LIN {X 0,Y 468.343,Z 264.353,A -85,B 0,C 180,E1 -7622.765,E2 -7622.765} C_VEL
LIN {X 0,Y 467.925,Z 273.797,A -85,B 0,C 180,E1 -7626.076,E2 -7626.076} C_VEL
LIN {X 0,Y 467.627,Z 283.274,A -85,B 0,C 180,E1 -7629.318,E2 -7629.318} C_VEL
LIN {X 0,Y 467.347,Z 292.793,A -85,B 0,C 180,E1 -7632.497,E2 -7632.497} C_VEL
LIN {X 0,Y 467.211,Z 299.063,A -85,B 0,C 180,E1 -7634.57,E2 -7634.57} C_VEL
LIN {X 0,Y 469.771,Z 314.339,A -85,B 0,C 180,E1 -7635.072,E2 -7635.072} C_VEL
LIN {X 0,Y 470.153,Z 319.57,A -85,B 0,C 180,E1 -7635.278,E2 -7635.278} C_VEL
LIN {X 0,Y 469.716,Z 331.244,A -85,B 0,C 180,E1 -7635.818,E2 -7635.818} C_VEL
LIN {X 0,Y 469.238,Z 342.474,A -85,B 0,C 180,E1 -7636.499,E2 -7636.499} C_VEL
LIN {X 0,Y 468.797,Z 353.368,A -85,B 0,C 180,E1 -7637.336,E2 -7637.336} C_VEL
LIN {X 0,Y 468.377,Z 363.596,A -85,B 0,C 180,E1 -7638.313,E2 -7638.313} C_VEL
LIN {X 0,Y 467.886,Z 372.785,A -85,B 0,C 180,E1 -7639.397,E2 -7639.397} C_VEL
LIN {X 0,Y 467.447,Z 381.688,A -85,B 0,C 180,E1 -7640.699,E2 -7640.699} C_VEL
LIN {X 0,Y 467.092,Z 388.849,A -85,B 0,C 180,E1 -7642,E2 -7642} C_VEL
LIN {X 0,Y 466.87,Z 395.224,A -85,B 0,C 180,E1 -7643.479,E2 -7643.479} C_VEL
LIN {X 0,Y 466.784,Z 399.677,A -85,B 0,C 180,E1 -7644.817,E2 -7644.817} C_VEL
LIN {X 0,Y 466.663,Z 401.958,A -85,B 0,C 180,E1 -7645.682,E2 -7645.682} C_VEL
LIN {X 0,Y 466.695,Z 403.807,A -85,B 0,C 180,E1 -7646.547,E2 -7646.547} C_VEL
LIN {X 0,Y 466.646,Z 405.193,A -85,B 0,C 180,E1 -7647.41,E2 -7647.41} C_VEL
LIN {X 0,Y 466.589,Z 406.785,A -85,B 0,C 180,E1 -7649.137,E2 -7649.137} C_VEL
LIN {X 0,Y 466.57,Z 407,A -85,B 0,C 180,E1 -7650,E2 -7650} C_VEL
LIN {X 0,Y 466.589,Z 406.786,A -85,B 0,C 180,E1 -7650.863,E2 -7650.863} C_VEL
LIN {X 0,Y 466.646,Z 405.195,A -85,B 0,C 180,E1 -7652.59,E2 -7652.59} C_VEL
LIN {X 0,Y 466.695,Z 403.81,A -85,B 0,C 180,E1 -7653.454,E2 -7653.454} C_VEL
LIN {X 0,Y 466.703,Z 400.895,A -85,B 0,C 180,E1 -7654.751,E2 -7654.751} C_VEL
LIN {X 0,Y 466.841,Z 396.947,A -85,B 0,C 180,E1 -7656.049,E2 -7656.049} C_VEL
LIN {X 0,Y 466.998,Z 390.874,A -85,B 0,C 180,E1 -7657.567,E2 -7657.567} C_VEL
LIN {X 0,Y 467.35,Z 384.234,A -85,B 0,C 180,E1 -7658.867,E2 -7658.867} C_VEL
LIN {X 0,Y 467.741,Z 375.991,A -85,B 0,C 180,E1 -7660.169,E2 -7660.169} C_VEL
LIN {X 0,Y 468.137,Z 367.516,A -85,B 0,C 180,E1 -7661.255,E2 -7661.255} C_VEL
LIN {X 0,Y 468.646,Z 357.189,A -85,B 0,C 180,E1 -7662.32,E2 -7662.32} C_VEL
LIN {X 0,Y 469.084,Z 345.563,A -85,B 0,C 180,E1 -7663.285,E2 -7663.285} C_VEL
LIN {X 0,Y 469.647,Z 333.231,A -85,B 0,C 180,E1 -7664.074,E2 -7664.074} C_VEL
LIN {X 0,Y 470.102,Z 320.858,A -85,B 0,C 180,E1 -7664.668,E2 -7664.668} C_VEL
LIN {X 0,Y 469.911,Z 315.479,A -85,B 0,C 180,E1 -7664.882,E2 -7664.882} C_VEL
LIN {X 0,Y 467.86,Z 303.142,A -85,B 0,C 180,E1 -7665.307,E2 -7665.307} C_VEL
LIN {X 0,Y 467.212,Z 298.992,A -85,B 0,C 180,E1 -7665.43,E2 -7665.43} C_VEL
LIN {X 0,Y 467.478,Z 289.113,A -85,B 0,C 180,E1 -7668.713,E2 -7668.713} C_VEL
LIN {X 0,Y 467.753,Z 279.15,A -85,B 0,C 180,E1 -7672.063,E2 -7672.063} C_VEL
LIN {X 0,Y 468.076,Z 269.794,A -85,B 0,C 180,E1 -7675.298,E2 -7675.298} C_VEL
LIN {X 0,Y 468.411,Z 261.608,A -85,B 0,C 180,E1 -7678.205,E2 -7678.205} C_VEL
LIN {X 0,Y 468.861,Z 252.156,A -85,B 0,C 180,E1 -7681.644,E2 -7681.644} C_VEL
LIN {X 0,Y 469.23,Z 244.096,A -85,B 0,C 180,E1 -7684.692,E2 -7684.692} C_VEL
LIN {X 0,Y 469.305,Z 240.672,A -85,B 0,C 180,E1 -7686.034,E2 -7686.034} C_VEL
LIN {X 0,Y 468.317,Z 234.357,A -85,B 0,C 180,E1 -7688.706,E2 -7688.706} C_VEL
LIN {X 0,Y 467.579,Z 230.247,A -85,B 0,C 180,E1 -7690.619,E2 -7690.619} C_VEL
LIN {X 0,Y 467.557,Z 230.25,A -85,B 0,C 180,E1 -7693.745,E2 -7693.745} C_VEL
LIN {X 0,Y 467.55,Z 230.244,A -85,B 0,C 180,E1 -7696.255,E2 -7696.255} C_VEL
LIN {X 0,Y 467.562,Z 230.24,A -85,B 0,C 180,E1 -7699.734,E2 -7699.734} C_VEL
LIN {X 0,Y 467.546,Z 230.246,A -85,B 0,C 180,E1 -7702.815,E2 -7702.815} C_VEL
LIN {X 0,Y 467.59,Z 230.241,A -85,B 0,C 180,E1 -7706.212,E2 -7706.212} C_VEL
LIN {X 0,Y 467.57,Z 230.242,A -85,B 0,C 180,E1 -7709.266,E2 -7709.266} C_VEL
LIN {X 0,Y 467.553,Z 230.247,A -85,B 0,C 180,E1 -7712.482,E2 -7712.482} C_VEL
LIN {X 0,Y 467.563,Z 230.241,A -85,B 0,C 180,E1 -7715.11,E2 -7715.11} C_VEL
LIN {X 0,Y 467.539,Z 230.249,A -85,B 0,C 180,E1 -7717.926,E2 -7717.926} C_VEL
LIN {X 0,Y 467.627,Z 230.236,A -85,B 0,C 180,E1 -7720.692,E2 -7720.692} C_VEL
LIN {X 0,Y 467.654,Z 230.234,A -85,B 0,C 180,E1 -7724.115,E2 -7724.115} C_VEL
LIN {X 0,Y 467.652,Z 230.233,A -85,B 0,C 180,E1 -7727.646,E2 -7727.646} C_VEL
LIN {X 0,Y 467.665,Z 230.232,A -85,B 0,C 180,E1 -7731.357,E2 -7731.357} C_VEL
LIN {X 0,Y 467.739,Z 230.222,A -85,B 0,C 180,E1 -7733.963,E2 -7733.963} C_VEL
LIN {X 0,Y 467.864,Z 230.206,A -85,B 0,C 180,E1 -7737.417,E2 -7737.417} C_VEL
LIN {X 0,Y 467.853,Z 230.207,A -85,B 0,C 180,E1 -7740,E2 -7740} C_VEL
LIN {X 0,Y 467.825,Z 230.208,A -85,B 0,C 180,E1 -7742.583,E2 -7742.583} C_VEL
LIN {X 0,Y 467.737,Z 230.221,A -85,B 0,C 180,E1 -7746.038,E2 -7746.038} C_VEL
LIN {X 0,Y 467.674,Z 230.231,A -85,B 0,C 180,E1 -7748.643,E2 -7748.643} C_VEL
LIN {X 0,Y 467.661,Z 230.231,A -85,B 0,C 180,E1 -7752.145,E2 -7752.145} C_VEL
LIN {X 0,Y 467.642,Z 230.232,A -85,B 0,C 180,E1 -7755.695,E2 -7755.695} C_VEL
LIN {X 0,Y 467.625,Z 230.235,A -85,B 0,C 180,E1 -7759.308,E2 -7759.308} C_VEL
LIN {X 0,Y 467.539,Z 230.246,A -85,B 0,C 180,E1 -7762.074,E2 -7762.074} C_VEL
LIN {X 0,Y 467.59,Z 230.241,A -85,B 0,C 180,E1 -7764.888,E2 -7764.888} C_VEL
LIN {X 0,Y 467.565,Z 230.243,A -85,B 0,C 180,E1 -7767.773,E2 -7767.773} C_VEL
LIN {X 0,Y 467.549,Z 230.244,A -85,B 0,C 180,E1 -7771.04,E2 -7771.04} C_VEL
LIN {X 0,Y 467.574,Z 230.241,A -85,B 0,C 180,E1 -7773.789,E2 -7773.789} C_VEL
LIN {X 0,Y 467.534,Z 230.248,A -85,B 0,C 180,E1 -7776.962,E2 -7776.962} C_VEL
LIN {X 0,Y 467.574,Z 230.242,A -85,B 0,C 180,E1 -7779.953,E2 -7779.953} C_VEL
LIN {X 0,Y 467.564,Z 230.245,A -85,B 0,C 180,E1 -7782.563,E2 -7782.563} C_VEL
LIN {X 0,Y 467.569,Z 230.24,A -85,B 0,C 180,E1 -7785.052,E2 -7785.052} C_VEL
LIN {X 0,Y 467.576,Z 230.241,A -85,B 0,C 180,E1 -7788.596,E2 -7788.596} C_VEL
LIN {X 0,Y 467.565,Z 230.243,A -85,B 0,C 180,E1 -7791.955,E2 -7791.955} C_VEL
LIN {X 0,Y 467.429,Z 230.261,A -85,B 0,C 180,E1 -7795.155,E2 -7795.155} C_VEL
LIN {X 0,Y 467.198,Z 230.291,A -85,B 0,C 180,E1 -7797.395,E2 -7797.395} C_VEL
LIN {X 0,Y 467.077,Z 232.866,A -85,B 0,C 180,E1 -7800.228,E2 -7800.228} C_VEL
LIN {X 0,Y 467.014,Z 235.784,A -85,B 0,C 180,E1 -7803.162,E2 -7803.162} C_VEL
LIN {X 0,Y 466.95,Z 238.685,A -85,B 0,C 180,E1 -7806.022,E2 -7806.022} C_VEL
LIN {X 0,Y 466.898,Z 241.727,A -85,B 0,C 180,E1 -7808.949,E2 -7808.949} C_VEL
LIN {X 0,Y 466.894,Z 244.613,A -85,B 0,C 180,E1 -7811.572,E2 -7811.572} C_VEL
LIN {X 0,Y 466.87,Z 247.359,A -85,B 0,C 180,E1 -7813.911,E2 -7813.911} C_VEL
LIN {X 0,Y 466.79,Z 248.655,A -85,B 0,C 180,E1 -7814.261,E2 -7814.261} C_VEL
LIN {X 0,Y 466.58,Z 251.014,A -85,B 0,C 180,E1 -7814.532,E2 -7814.532} C_VEL
LIN {X 0,Y 466.15,Z 255.079,A -85,B 0,C 180,E1 -7814.785,E2 -7814.785} C_VEL
LIN {X 0,Y 463.561,Z 272.449,A -85,B 0,C 180,E1 -7815.439,E2 -7815.439} C_VEL
LIN {X 0,Y 463.282,Z 275.826,A -85,B 0,C 180,E1 -7815.608,E2 -7815.608} C_VEL
LIN {X 0,Y 462.831,Z 287.027,A -85,B 0,C 180,E1 -7816.291,E2 -7816.291} C_VEL
LIN {X 0,Y 462.369,Z 298.125,A -85,B 0,C 180,E1 -7817.156,E2 -7817.156} C_VEL
LIN {X 0,Y 461.823,Z 308.332,A -85,B 0,C 180,E1 -7818.144,E2 -7818.144} C_VEL
LIN {X 0,Y 461.343,Z 317.483,A -85,B 0,C 180,E1 -7819.245,E2 -7819.245} C_VEL
LIN {X 0,Y 460.871,Z 326.359,A -85,B 0,C 180,E1 -7820.565,E2 -7820.565} C_VEL
LIN {X 0,Y 460.435,Z 333.504,A -85,B 0,C 180,E1 -7821.883,E2 -7821.883} C_VEL
LIN {X 0,Y 460.182,Z 339.823,A -85,B 0,C 180,E1 -7823.373,E2 -7823.373} C_VEL
LIN {X 0,Y 459.847,Z 344.308,A -85,B 0,C 180,E1 -7824.738,E2 -7824.738} C_VEL
LIN {X 0,Y 459.919,Z 346.57,A -85,B 0,C 180,E1 -7825.618,E2 -7825.618} C_VEL
LIN {X 0,Y 459.824,Z 348.421,A -85,B 0,C 180,E1 -7826.495,E2 -7826.495} C_VEL
LIN {X 0,Y 459.781,Z 349.815,A -85,B 0,C 180,E1 -7827.372,E2 -7827.372} C_VEL
LIN {X 0,Y 459.567,Z 351.426,A -85,B 0,C 180,E1 -7829.124,E2 -7829.124} C_VEL
LIN {X 0,Y 459.55,Z 351.66,A -85,B 0,C 180,E1 -7830,E2 -7830} C_VEL
LIN {X 0,Y 459.642,Z 350.892,A -85,B 0,C 180,E1 -7831.752,E2 -7831.752} C_VEL
LIN {X 0,Y 459.781,Z 349.928,A -85,B 0,C 180,E1 -7832.628,E2 -7832.628} C_VEL
LIN {X 0,Y 459.823,Z 348.583,A -85,B 0,C 180,E1 -7833.505,E2 -7833.505} C_VEL
LIN {X 0,Y 459.903,Z 345.741,A -85,B 0,C 180,E1 -7834.821,E2 -7834.821} C_VEL
LIN {X 0,Y 460.044,Z 341.884,A -85,B 0,C 180,E1 -7836.139,E2 -7836.139} C_VEL
LIN {X 0,Y 460.253,Z 336.906,A -85,B 0,C 180,E1 -7837.458,E2 -7837.458} C_VEL
LIN {X 0,Y 460.598,Z 330.632,A -85,B 0,C 180,E1 -7838.777,E2 -7838.777} C_VEL
LIN {X 0,Y 461.004,Z 322.776,A -85,B 0,C 180,E1 -7840.097,E2 -7840.097} C_VEL
LIN {X 0,Y 461.527,Z 314.755,A -85,B 0,C 180,E1 -7841.195,E2 -7841.195} C_VEL
LIN {X 0,Y 462,Z 304.971,A -85,B 0,C 180,E1 -7842.296,E2 -7842.296} C_VEL
LIN {X 0,Y 462.475,Z 295.336,A -85,B 0,C 180,E1 -7843.176,E2 -7843.176} C_VEL
LIN {X 0,Y 462.937,Z 284.671,A -85,B 0,C 180,E1 -7843.961,E2 -7843.961} C_VEL
LIN {X 0,Y 463.391,Z 272.342,A -85,B 0,C 180,E1 -7844.66,E2 -7844.66} C_VEL
LIN {X 0,Y 463.563,Z 264.842,A -85,B 0,C 180,E1 -7844.998,E2 -7844.998} C_VEL
LIN {X 0,Y 460.782,Z 252.445,A -85,B 0,C 180,E1 -7845.514,E2 -7845.514} C_VEL
LIN {X 0,Y 459.861,Z 248.614,A -85,B 0,C 180,E1 -7845.671,E2 -7845.671} C_VEL
LIN {X 0,Y 459.83,Z 245.097,A -85,B 0,C 180,E1 -7848.721,E2 -7848.721} C_VEL
LIN {X 0,Y 459.836,Z 242.04,A -85,B 0,C 180,E1 -7851.519,E2 -7851.519} C_VEL
LIN {X 0,Y 459.903,Z 239.086,A -85,B 0,C 180,E1 -7854.368,E2 -7854.368} C_VEL
LIN {X 0,Y 459.989,Z 235.815,A -85,B 0,C 180,E1 -7857.605,E2 -7857.605} C_VEL
LIN {X 0,Y 460.045,Z 233.208,A -85,B 0,C 180,E1 -7860.274,E2 -7860.274} C_VEL
LIN {X 0,Y 460.081,Z 231.215,A -85,B 0,C 180,E1 -7862.32,E2 -7862.32} C_VEL
LIN {X 0,Y 460.428,Z 231.131,A -85,B 0,C 180,E1 -7865.453,E2 -7865.453} C_VEL
LIN {X 0,Y 460.52,Z 231.122,A -85,B 0,C 180,E1 -7868.734,E2 -7868.734} C_VEL
LIN {X 0,Y 460.52,Z 231.12,A -85,B 0,C 180,E1 -7871.6,E2 -7871.6} C_VEL
LIN {X 0,Y 460.514,Z 231.12,A -85,B 0,C 180,E1 -7874.589,E2 -7874.589} C_VEL
LIN {X 0,Y 460.506,Z 231.124,A -85,B 0,C 180,E1 -7877.816,E2 -7877.816} C_VEL
LIN {X 0,Y 460.534,Z 231.119,A -85,B 0,C 180,E1 -7881.104,E2 -7881.104} C_VEL
LIN {X 0,Y 460.511,Z 231.121,A -85,B 0,C 180,E1 -7884.554,E2 -7884.554} C_VEL
LIN {X 0,Y 460.532,Z 231.122,A -85,B 0,C 180,E1 -7887.715,E2 -7887.715} C_VEL
LIN {X 0,Y 460.523,Z 231.119,A -85,B 0,C 180,E1 -7890.768,E2 -7890.768} C_VEL
LIN {X 0,Y 460.534,Z 231.119,A -85,B 0,C 180,E1 -7893.733,E2 -7893.733} C_VEL
LIN {X 0,Y 460.547,Z 231.118,A -85,B 0,C 180,E1 -7896.624,E2 -7896.624} C_VEL
LIN {X 0,Y 460.554,Z 231.12,A -85,B 0,C 180,E1 -7899.453,E2 -7899.453} C_VEL
LIN {X 0,Y 460.543,Z 231.115,A -85,B 0,C 180,E1 -7902.229,E2 -7902.229} C_VEL
LIN {X 0,Y 460.561,Z 231.119,A -85,B 0,C 180,E1 -7904.965,E2 -7904.965} C_VEL
LIN {X 0,Y 460.615,Z 231.111,A -85,B 0,C 180,E1 -7908.559,E2 -7908.559} C_VEL
LIN {X 0,Y 460.699,Z 231.099,A -85,B 0,C 180,E1 -7912.109,E2 -7912.109} C_VEL
LIN {X 0,Y 460.691,Z 231.101,A -85,B 0,C 180,E1 -7914.748,E2 -7914.748} C_VEL
LIN {X 0,Y 460.769,Z 231.087,A -85,B 0,C 180,E1 -7917.377,E2 -7917.377} C_VEL
LIN {X 0,Y 460.821,Z 231.083,A -85,B 0,C 180,E1 -7920,E2 -7920} C_VEL
LIN {X 0,Y 460.803,Z 231.086,A -85,B 0,C 180,E1 -7922.622,E2 -7922.622} C_VEL
LIN {X 0,Y 460.703,Z 231.098,A -85,B 0,C 180,E1 -7926.13,E2 -7926.13} C_VEL
LIN {X 0,Y 460.618,Z 231.109,A -85,B 0,C 180,E1 -7928.776,E2 -7928.776} C_VEL
LIN {X 0,Y 460.599,Z 231.111,A -85,B 0,C 180,E1 -7932.435,E2 -7932.435} C_VEL
LIN {X 0,Y 460.603,Z 231.112,A -85,B 0,C 180,E1 -7935.997,E2 -7935.997} C_VEL
LIN {X 0,Y 460.574,Z 231.114,A -85,B 0,C 180,E1 -7938.902,E2 -7938.902} C_VEL
LIN {X 0,Y 460.519,Z 231.121,A -85,B 0,C 180,E1 -7941.486,E2 -7941.486} C_VEL
LIN {X 0,Y 460.52,Z 231.12,A -85,B 0,C 180,E1 -7944.334,E2 -7944.334} C_VEL
LIN {X 0,Y 460.493,Z 231.123,A -85,B 0,C 180,E1 -7947.249,E2 -7947.249} C_VEL
LIN {X 0,Y 460.506,Z 231.122,A -85,B 0,C 180,E1 -7950.24,E2 -7950.24} C_VEL
LIN {X 0,Y 460.531,Z 231.12,A -85,B 0,C 180,E1 -7953.325,E2 -7953.325} C_VEL
LIN {X 0,Y 460.474,Z 231.126,A -85,B 0,C 180,E1 -7956.53,E2 -7956.53} C_VEL
LIN {X 0,Y 460.515,Z 231.123,A -85,B 0,C 180,E1 -7959.864,E2 -7959.864} C_VEL
LIN {X 0,Y 460.481,Z 231.129,A -85,B 0,C 180,E1 -7962.896,E2 -7962.896} C_VEL
LIN {X 0,Y 460.511,Z 231.123,A -85,B 0,C 180,E1 -7965.831,E2 -7965.831} C_VEL
LIN {X 0,Y 460.567,Z 231.239,A -85,B 0,C 180,E1 -7969.188,E2 -7969.188} C_VEL
LIN {X 0,Y 461.887,Z 238.631,A -85,B 0,C 180,E1 -7972.509,E2 -7972.509} C_VEL
LIN {X 0,Y 462.343,Z 242.67,A -85,B 0,C 180,E1 -7974.208,E2 -7974.208} C_VEL
LIN {X 0,Y 462.056,Z 249.276,A -85,B 0,C 180,E1 -7976.799,E2 -7976.799} C_VEL
LIN {X 0,Y 461.603,Z 257.362,A -85,B 0,C 180,E1 -7979.839,E2 -7979.839} C_VEL
LIN {X 0,Y 461.29,Z 265.482,A -85,B 0,C 180,E1 -7982.802,E2 -7982.802} C_VEL
LIN {X 0,Y 460.862,Z 275.008,A -85,B 0,C 180,E1 -7986.203,E2 -7986.203} C_VEL
LIN {X 0,Y 460.612,Z 283.015,A -85,B 0,C 180,E1 -7988.995,E2 -7988.995} C_VEL
LIN {X 0,Y 460.304,Z 292.453,A -85,B 0,C 180,E1 -7992.22,E2 -7992.22} C_VEL
LIN {X 0,Y 460.163,Z 298.721,A -85,B 0,C 180,E1 -7994.339,E2 -7994.339} C_VEL
LIN {X 0,Y 462.555,Z 313.328,A -85,B 0,C 180,E1 -7994.813,E2 -7994.813} C_VEL
LIN {X 0,Y 463.269,Z 319.141,A -85,B 0,C 180,E1 -7995.055,E2 -7995.055} C_VEL
LIN {X 0,Y 462.821,Z 330.815,A -85,B 0,C 180,E1 -7995.602,E2 -7995.602} C_VEL
LIN {X 0,Y 462.265,Z 343.158,A -85,B 0,C 180,E1 -7996.37,E2 -7996.37} C_VEL
LIN {X 0,Y 461.79,Z 353.56,A -85,B 0,C 180,E1 -7997.195,E2 -7997.195} C_VEL
LIN {X 0,Y 461.369,Z 363.164,A -85,B 0,C 180,E1 -7998.133,E2 -7998.133} C_VEL
LIN {X 0,Y 460.873,Z 372.383,A -85,B 0,C 180,E1 -7999.234,E2 -7999.234} C_VEL
LIN {X 0,Y 460.417,Z 381.373,A -85,B 0,C 180,E1 -8000.556,E2 -8000.556} C_VEL
LIN {X 0,Y 460.054,Z 388.612,A -85,B 0,C 180,E1 -8001.877,E2 -8001.877} C_VEL
LIN {X 0,Y 459.848,Z 393.503,A -85,B 0,C 180,E1 -8002.977,E2 -8002.977} C_VEL
LIN {X 0,Y 459.756,Z 398.263,A -85,B 0,C 180,E1 -8004.298,E2 -8004.298} C_VEL
LIN {X 0,Y 459.579,Z 401.895,A -85,B 0,C 180,E1 -8005.615,E2 -8005.615} C_VEL
LIN {X 0,Y 459.591,Z 403.773,A -85,B 0,C 180,E1 -8006.493,E2 -8006.493} C_VEL
LIN {X 0,Y 459.57,Z 405.175,A -85,B 0,C 180,E1 -8007.371,E2 -8007.371} C_VEL
LIN {X 0,Y 459.494,Z 406.779,A -85,B 0,C 180,E1 -8009.124,E2 -8009.124} C_VEL
LIN {X 0,Y 459.474,Z 406.994,A -85,B 0,C 180,E1 -8010,E2 -8010} C_VEL
LIN {X 0,Y 459.494,Z 406.779,A -85,B 0,C 180,E1 -8010.877,E2 -8010.877} C_VEL
LIN {X 0,Y 459.57,Z 405.178,A -85,B 0,C 180,E1 -8012.63,E2 -8012.63} C_VEL
LIN {X 0,Y 459.591,Z 403.776,A -85,B 0,C 180,E1 -8013.507,E2 -8013.507} C_VEL
LIN {X 0,Y 459.635,Z 400.818,A -85,B 0,C 180,E1 -8014.824,E2 -8014.824} C_VEL
LIN {X 0,Y 459.758,Z 396.816,A -85,B 0,C 180,E1 -8016.143,E2 -8016.143} C_VEL
LIN {X 0,Y 459.929,Z 390.661,A -85,B 0,C 180,E1 -8017.684,E2 -8017.684} C_VEL
LIN {X 0,Y 460.288,Z 383.947,A -85,B 0,C 180,E1 -8019.004,E2 -8019.004} C_VEL
LIN {X 0,Y 460.705,Z 375.618,A -85,B 0,C 180,E1 -8020.326,E2 -8020.326} C_VEL
LIN {X 0,Y 461.141,Z 367.087,A -85,B 0,C 180,E1 -8021.428,E2 -8021.428} C_VEL
LIN {X 0,Y 461.65,Z 356.929,A -85,B 0,C 180,E1 -8022.494,E2 -8022.494} C_VEL
LIN {X 0,Y 462.108,Z 346.136,A -85,B 0,C 180,E1 -8023.411,E2 -8023.411} C_VEL
LIN {X 0,Y 462.655,Z 334.731,A -85,B 0,C 180,E1 -8024.179,E2 -8024.179} C_VEL
LIN {X 0,Y 463.137,Z 323.038,A -85,B 0,C 180,E1 -8024.781,E2 -8024.781} C_VEL
LIN {X 0,Y 463.005,Z 316.628,A -85,B 0,C 180,E1 -8025.051,E2 -8025.051} C_VEL
LIN {X 0,Y 460.944,Z 303.952,A -85,B 0,C 180,E1 -8025.512,E2 -8025.512} C_VEL
LIN {X 0,Y 460.149,Z 298.542,A -85,B 0,C 180,E1 -8025.676,E2 -8025.676} C_VEL
LIN {X 0,Y 460.447,Z 288.283,A -85,B 0,C 180,E1 -8029.178,E2 -8029.178} C_VEL
LIN {X 0,Y 460.73,Z 278.884,A -85,B 0,C 180,E1 -8032.418,E2 -8032.418} C_VEL
LIN {X 0,Y 461.117,Z 268.93,A -85,B 0,C 180,E1 -8035.942,E2 -8035.942} C_VEL
LIN {X 0,Y 461.428,Z 261.387,A -85,B 0,C 180,E1 -8038.671,E2 -8038.671} C_VEL
LIN {X 0,Y 461.824,Z 253.615,A -85,B 0,C 180,E1 -8041.548,E2 -8041.548} C_VEL
LIN {X 0,Y 462.191,Z 246.577,A -85,B 0,C 180,E1 -8044.237,E2 -8044.237} C_VEL
LIN {X 0,Y 462.24,Z 241.251,A -85,B 0,C 180,E1 -8046.368,E2 -8046.368} C_VEL
LIN {X 0,Y 461.256,Z 235.171,A -85,B 0,C 180,E1 -8049.007,E2 -8049.007} C_VEL
LIN {X 0,Y 460.551,Z 231.121,A -85,B 0,C 180,E1 -8050.912,E2 -8050.912} C_VEL
LIN {X 0,Y 460.512,Z 231.126,A -85,B 0,C 180,E1 -8054.17,E2 -8054.17} C_VEL
LIN {X 0,Y 460.483,Z 231.129,A -85,B 0,C 180,E1 -8057.104,E2 -8057.104} C_VEL
LIN {X 0,Y 460.516,Z 231.119,A -85,B 0,C 180,E1 -8060.136,E2 -8060.136} C_VEL
LIN {X 0,Y 460.476,Z 231.125,A -85,B 0,C 180,E1 -8063.47,E2 -8063.47} C_VEL
LIN {X 0,Y 460.533,Z 231.12,A -85,B 0,C 180,E1 -8066.675,E2 -8066.675} C_VEL
LIN {X 0,Y 460.508,Z 231.122,A -85,B 0,C 180,E1 -8069.76,E2 -8069.76} C_VEL
LIN {X 0,Y 460.494,Z 231.123,A -85,B 0,C 180,E1 -8072.751,E2 -8072.751} C_VEL
LIN {X 0,Y 460.521,Z 231.12,A -85,B 0,C 180,E1 -8075.667,E2 -8075.667} C_VEL
LIN {X 0,Y 460.526,Z 231.12,A -85,B 0,C 180,E1 -8078.578,E2 -8078.578} C_VEL
LIN {X 0,Y 460.591,Z 231.112,A -85,B 0,C 180,E1 -8081.311,E2 -8081.311} C_VEL
LIN {X 0,Y 460.609,Z 231.111,A -85,B 0,C 180,E1 -8084.059,E2 -8084.059} C_VEL
LIN {X 0,Y 460.607,Z 231.111,A -85,B 0,C 180,E1 -8087.666,E2 -8087.666} C_VEL
LIN {X 0,Y 460.612,Z 231.109,A -85,B 0,C 180,E1 -8091.224,E2 -8091.224} C_VEL
LIN {X 0,Y 460.705,Z 231.098,A -85,B 0,C 180,E1 -8093.87,E2 -8093.87} C_VEL
LIN {X 0,Y 460.804,Z 231.086,A -85,B 0,C 180,E1 -8097.378,E2 -8097.378} C_VEL
LIN {X 0,Y 460.823,Z 231.083,A -85,B 0,C 180,E1 -8100,E2 -8100} C_VEL
LIN {X 0,Y 460.77,Z 231.087,A -85,B 0,C 180,E1 -8102.623,E2 -8102.623} C_VEL
LIN {X 0,Y 460.702,Z 231.097,A -85,B 0,C 180,E1 -8106.13,E2 -8106.13} C_VEL
LIN {X 0,Y 460.624,Z 231.11,A -85,B 0,C 180,E1 -8108.776,E2 -8108.776} C_VEL
LIN {X 0,Y 460.615,Z 231.109,A -85,B 0,C 180,E1 -8112.334,E2 -8112.334} C_VEL
LIN {X 0,Y 460.583,Z 231.11,A -85,B 0,C 180,E1 -8115.988,E2 -8115.988} C_VEL
LIN {X 0,Y 460.571,Z 231.113,A -85,B 0,C 180,E1 -8119.616,E2 -8119.616} C_VEL
LIN {X 0,Y 460.516,Z 231.124,A -85,B 0,C 180,E1 -8122.429,E2 -8122.429} C_VEL
LIN {X 0,Y 460.554,Z 231.116,A -85,B 0,C 180,E1 -8125.797,E2 -8125.797} C_VEL
LIN {X 0,Y 460.517,Z 231.121,A -85,B 0,C 180,E1 -8128.235,E2 -8128.235} C_VEL
LIN {X 0,Y 460.524,Z 231.117,A -85,B 0,C 180,E1 -8131.282,E2 -8131.282} C_VEL
LIN {X 0,Y 460.527,Z 231.121,A -85,B 0,C 180,E1 -8134.504,E2 -8134.504} C_VEL
LIN {X 0,Y 460.505,Z 231.123,A -85,B 0,C 180,E1 -8137.623,E2 -8137.623} C_VEL
LIN {X 0,Y 460.539,Z 231.119,A -85,B 0,C 180,E1 -8140.268,E2 -8140.268} C_VEL
LIN {X 0,Y 460.512,Z 231.121,A -85,B 0,C 180,E1 -8143.374,E2 -8143.374} C_VEL
LIN {X 0,Y 460.512,Z 231.12,A -85,B 0,C 180,E1 -8146.625,E2 -8146.625} C_VEL
LIN {X 0,Y 460.538,Z 231.121,A -85,B 0,C 180,E1 -8149.732,E2 -8149.732} C_VEL
LIN {X 0,Y 460.498,Z 231.124,A -85,B 0,C 180,E1 -8152.525,E2 -8152.525} C_VEL
LIN {X 0,Y 460.352,Z 231.145,A -85,B 0,C 180,E1 -8155.607,E2 -8155.607} C_VEL
LIN {X 0,Y 460.092,Z 231.177,A -85,B 0,C 180,E1 -8157.681,E2 -8157.681} C_VEL
LIN {X 0,Y 460.046,Z 234.114,A -85,B 0,C 180,E1 -8160.734,E2 -8160.734} C_VEL
LIN {X 0,Y 459.928,Z 237.074,A -85,B 0,C 180,E1 -8163.695,E2 -8163.695} C_VEL
LIN {X 0,Y 459.878,Z 239.966,A -85,B 0,C 180,E1 -8166.588,E2 -8166.588} C_VEL
LIN {X 0,Y 459.823,Z 242.938,A -85,B 0,C 180,E1 -8169.418,E2 -8169.418} C_VEL
LIN {X 0,Y 459.811,Z 246.022,A -85,B 0,C 180,E1 -8172.2,E2 -8172.2} C_VEL
LIN {X 0,Y 459.86,Z 248.691,A -85,B 0,C 180,E1 -8174.445,E2 -8174.445} C_VEL
LIN {X 0,Y 463.035,Z 262.336,A -85,B 0,C 180,E1 -8174.98,E2 -8174.98} C_VEL
LIN {X 0,Y 463.574,Z 265.423,A -85,B 0,C 180,E1 -8175.121,E2 -8175.121} C_VEL
LIN {X 0,Y 463.282,Z 275.826,A -85,B 0,C 180,E1 -8175.608,E2 -8175.608} C_VEL
LIN {X 0,Y 462.431,Z 281.281,A -85,B 0,C 180,E1 -8175.896,E2 -8175.896} C_VEL
LIN {X 0,Y 457.843,Z 293.207,A -85,B 0,C 180,E1 -8176.581,E2 -8176.581} C_VEL
LIN {X 0,Y 455.662,Z 299.718,A -85,B 0,C 180,E1 -8177.067,E2 -8177.067} C_VEL
LIN {X 0,Y 455.236,Z 302.818,A -85,B 0,C 180,E1 -8177.352,E2 -8177.352} C_VEL
LIN {X 0,Y 454.693,Z 312.65,A -85,B 0,C 180,E1 -8178.408,E2 -8178.408} C_VEL
LIN {X 0,Y 454.202,Z 321.118,A -85,B 0,C 180,E1 -8179.525,E2 -8179.525} C_VEL
LIN {X 0,Y 453.717,Z 329.337,A -85,B 0,C 180,E1 -8180.864,E2 -8180.864} C_VEL
LIN {X 0,Y 453.38,Z 334.959,A -85,B 0,C 180,E1 -8181.98,E2 -8181.98} C_VEL
LIN {X 0,Y 453.141,Z 340.484,A -85,B 0,C 180,E1 -8183.335,E2 -8183.335} C_VEL
LIN {X 0,Y 452.786,Z 344.736,A -85,B 0,C 180,E1 -8184.656,E2 -8184.656} C_VEL
LIN {X 0,Y 452.85,Z 346.998,A -85,B 0,C 180,E1 -8185.549,E2 -8185.549} C_VEL
LIN {X 0,Y 452.759,Z 348.849,A -85,B 0,C 180,E1 -8186.44,E2 -8186.44} C_VEL
LIN {X 0,Y 452.71,Z 350.242,A -85,B 0,C 180,E1 -8187.33,E2 -8187.33} C_VEL
LIN {X 0,Y 452.502,Z 351.852,A -85,B 0,C 180,E1 -8189.11,E2 -8189.11} C_VEL
LIN {X 0,Y 452.482,Z 352.086,A -85,B 0,C 180,E1 -8190,E2 -8190} C_VEL
LIN {X 0,Y 452.584,Z 351.317,A -85,B 0,C 180,E1 -8191.78,E2 -8191.78} C_VEL
LIN {X 0,Y 452.697,Z 350.354,A -85,B 0,C 180,E1 -8192.669,E2 -8192.669} C_VEL
LIN {X 0,Y 452.758,Z 349.009,A -85,B 0,C 180,E1 -8193.56,E2 -8193.56} C_VEL
LIN {X 0,Y 452.845,Z 346.167,A -85,B 0,C 180,E1 -8194.897,E2 -8194.897} C_VEL
LIN {X 0,Y 453.009,Z 342.309,A -85,B 0,C 180,E1 -8196.234,E2 -8196.234} C_VEL
LIN {X 0,Y 453.222,Z 337.331,A -85,B 0,C 180,E1 -8197.574,E2 -8197.574} C_VEL
LIN {X 0,Y 453.61,Z 331.056,A -85,B 0,C 180,E1 -8198.913,E2 -8198.913} C_VEL
LIN {X 0,Y 454.038,Z 323.199,A -85,B 0,C 180,E1 -8200.254,E2 -8200.254} C_VEL
LIN {X 0,Y 454.578,Z 315.178,A -85,B 0,C 180,E1 -8201.369,E2 -8201.369} C_VEL
LIN {X 0,Y 455.078,Z 305.393,A -85,B 0,C 180,E1 -8202.486,E2 -8202.486} C_VEL
LIN {X 0,Y 455.645,Z 294.238,A -85,B 0,C 180,E1 -8203.502,E2 -8203.502} C_VEL
LIN {X 0,Y 456.192,Z 281.819,A -85,B 0,C 180,E1 -8204.384,E2 -8204.384} C_VEL
LIN {X 0,Y 456.625,Z 269.276,A -85,B 0,C 180,E1 -8205.054,E2 -8205.054} C_VEL
LIN {X 0,Y 456.601,Z 265.287,A -85,B 0,C 180,E1 -8205.231,E2 -8205.231} C_VEL
LIN {X 0,Y 453.639,Z 252.524,A -85,B 0,C 180,E1 -8205.773,E2 -8205.773} C_VEL
LIN {X 0,Y 452.789,Z 249.043,A -85,B 0,C 180,E1 -8205.905,E2 -8205.905} C_VEL
LIN {X 0,Y 452.765,Z 245.471,A -85,B 0,C 180,E1 -8209.024,E2 -8209.024} C_VEL
LIN {X 0,Y 452.776,Z 242.386,A -85,B 0,C 180,E1 -8211.872,E2 -8211.872} C_VEL
LIN {X 0,Y 452.868,Z 239.405,A -85,B 0,C 180,E1 -8214.772,E2 -8214.772} C_VEL
LIN {X 0,Y 452.934,Z 236.349,A -85,B 0,C 180,E1 -8217.816,E2 -8217.816} C_VEL
LIN {X 0,Y 452.986,Z 233.469,A -85,B 0,C 180,E1 -8220.796,E2 -8220.796} C_VEL
LIN {X 0,Y 453.015,Z 232.459,A -85,B 0,C 180,E1 -8221.835,E2 -8221.835} C_VEL
LIN {X 0,Y 453.161,Z 232.041,A -85,B 0,C 180,E1 -8223.125,E2 -8223.125} C_VEL
LIN {X 0,Y 453.411,Z 232.008,A -85,B 0,C 180,E1 -8226.087,E2 -8226.087} C_VEL
LIN {X 0,Y 453.472,Z 231.998,A -85,B 0,C 180,E1 -8229.203,E2 -8229.203} C_VEL
LIN {X 0,Y 453.461,Z 232.001,A -85,B 0,C 180,E1 -8231.932,E2 -8231.932} C_VEL
LIN {X 0,Y 453.484,Z 231.996,A -85,B 0,C 180,E1 -8235.471,E2 -8235.471} C_VEL
LIN {X 0,Y 453.465,Z 232,A -85,B 0,C 180,E1 -8238.207,E2 -8238.207} C_VEL
LIN {X 0,Y 453.471,Z 231.998,A -85,B 0,C 180,E1 -8240.797,E2 -8240.797} C_VEL
LIN {X 0,Y 453.457,Z 232.003,A -85,B 0,C 180,E1 -8243.917,E2 -8243.917} C_VEL
LIN {X 0,Y 453.481,Z 231.996,A -85,B 0,C 180,E1 -8247.151,E2 -8247.151} C_VEL
LIN {X 0,Y 453.464,Z 231.998,A -85,B 0,C 180,E1 -8250.267,E2 -8250.267} C_VEL
LIN {X 0,Y 453.467,Z 232.001,A -85,B 0,C 180,E1 -8253.291,E2 -8253.291} C_VEL
LIN {X 0,Y 453.499,Z 231.995,A -85,B 0,C 180,E1 -8256.238,E2 -8256.238} C_VEL
LIN {X 0,Y 453.485,Z 231.998,A -85,B 0,C 180,E1 -8259.118,E2 -8259.118} C_VEL
LIN {X 0,Y 453.499,Z 231.993,A -85,B 0,C 180,E1 -8261.944,E2 -8261.944} C_VEL
LIN {X 0,Y 453.533,Z 231.992,A -85,B 0,C 180,E1 -8264.726,E2 -8264.726} C_VEL
LIN {X 0,Y 453.563,Z 231.988,A -85,B 0,C 180,E1 -8268.379,E2 -8268.379} C_VEL
LIN {X 0,Y 453.655,Z 231.975,A -85,B 0,C 180,E1 -8271.985,E2 -8271.985} C_VEL
LIN {X 0,Y 453.665,Z 231.976,A -85,B 0,C 180,E1 -8274.667,E2 -8274.667} C_VEL
LIN {X 0,Y 453.693,Z 231.971,A -85,B 0,C 180,E1 -8278.225,E2 -8278.225} C_VEL
LIN {X 0,Y 453.791,Z 231.958,A -85,B 0,C 180,E1 -8280,E2 -8280} C_VEL
LIN {X 0,Y 453.747,Z 231.965,A -85,B 0,C 180,E1 -8282.663,E2 -8282.663} C_VEL
LIN {X 0,Y 453.67,Z 231.974,A -85,B 0,C 180,E1 -8286.225,E2 -8286.225} C_VEL
LIN {X 0,Y 453.583,Z 231.984,A -85,B 0,C 180,E1 -8288.914,E2 -8288.914} C_VEL
LIN {X 0,Y 453.567,Z 231.986,A -85,B 0,C 180,E1 -8292.529,E2 -8292.529} C_VEL
LIN {X 0,Y 453.548,Z 231.99,A -85,B 0,C 180,E1 -8296.196,E2 -8296.196} C_VEL
LIN {X 0,Y 453.523,Z 231.992,A -85,B 0,C 180,E1 -8299.041,E2 -8299.041} C_VEL
LIN {X 0,Y 453.479,Z 231.999,A -85,B 0,C 180,E1 -8301.836,E2 -8301.836} C_VEL
LIN {X 0,Y 453.471,Z 231.996,A -85,B 0,C 180,E1 -8304.737,E2 -8304.737} C_VEL
LIN {X 0,Y 453.465,Z 232,A -85,B 0,C 180,E1 -8307.943,E2 -8307.943} C_VEL
LIN {X 0,Y 453.476,Z 231.997,A -85,B 0,C 180,E1 -8310.76,E2 -8310.76} C_VEL
LIN {X 0,Y 453.479,Z 232,A -85,B 0,C 180,E1 -8313.913,E2 -8313.913} C_VEL
LIN {X 0,Y 453.451,Z 232.002,A -85,B 0,C 180,E1 -8317.19,E2 -8317.19} C_VEL
LIN {X 0,Y 453.472,Z 231.996,A -85,B 0,C 180,E1 -8320.612,E2 -8320.612} C_VEL
LIN {X 0,Y 453.461,Z 232.001,A -85,B 0,C 180,E1 -8324.222,E2 -8324.222} C_VEL
LIN {X 0,Y 453.465,Z 232.002,A -85,B 0,C 180,E1 -8327.005,E2 -8327.005} C_VEL
LIN {X 0,Y 453.537,Z 232.148,A -85,B 0,C 180,E1 -8328.89,E2 -8328.89} C_VEL
LIN {X 0,Y 454.748,Z 238.96,A -85,B 0,C 180,E1 -8332.017,E2 -8332.017} C_VEL
LIN {X 0,Y 455.35,Z 243.762,A -85,B 0,C 180,E1 -8334.091,E2 -8334.091} C_VEL
LIN {X 0,Y 455.091,Z 249.795,A -85,B 0,C 180,E1 -8336.504,E2 -8336.504} C_VEL
LIN {X 0,Y 454.696,Z 257.143,A -85,B 0,C 180,E1 -8339.332,E2 -8339.332} C_VEL
LIN {X 0,Y 454.262,Z 266.614,A -85,B 0,C 180,E1 -8342.845,E2 -8342.845} C_VEL
LIN {X 0,Y 453.809,Z 275.999,A -85,B 0,C 180,E1 -8346.256,E2 -8346.256} C_VEL
LIN {X 0,Y 453.46,Z 285.422,A -85,B 0,C 180,E1 -8349.591,E2 -8349.591} C_VEL
LIN {X 0,Y 453.188,Z 293.411,A -85,B 0,C 180,E1 -8352.398,E2 -8352.398} C_VEL
LIN {X 0,Y 453.084,Z 298.359,A -85,B 0,C 180,E1 -8354.095,E2 -8354.095} C_VEL
LIN {X 0,Y 455.261,Z 311.681,A -85,B 0,C 180,E1 -8354.523,E2 -8354.523} C_VEL
LIN {X 0,Y 456.336,Z 320.016,A -85,B 0,C 180,E1 -8354.879,E2 -8354.879} C_VEL
LIN {X 0,Y 455.821,Z 332.38,A -85,B 0,C 180,E1 -8355.49,E2 -8355.49} C_VEL
LIN {X 0,Y 455.249,Z 344.273,A -85,B 0,C 180,E1 -8356.27,E2 -8356.27} C_VEL
LIN {X 0,Y 454.728,Z 355.079,A -85,B 0,C 180,E1 -8357.177,E2 -8357.177} C_VEL
LIN {X 0,Y 454.272,Z 364.701,A -85,B 0,C 180,E1 -8358.171,E2 -8358.171} C_VEL
LIN {X 0,Y 453.735,Z 373.592,A -85,B 0,C 180,E1 -8359.288,E2 -8359.288} C_VEL
LIN {X 0,Y 453.31,Z 382.274,A -85,B 0,C 180,E1 -8360.631,E2 -8360.631} C_VEL
LIN {X 0,Y 452.924,Z 389.214,A -85,B 0,C 180,E1 -8361.972,E2 -8361.972} C_VEL
LIN {X 0,Y 452.71,Z 395.438,A -85,B 0,C 180,E1 -8363.493,E2 -8363.493} C_VEL
LIN {X 0,Y 452.567,Z 400.39,A -85,B 0,C 180,E1 -8365.1,E2 -8365.1} C_VEL
LIN {X 0,Y 452.493,Z 403.346,A -85,B 0,C 180,E1 -8366.438,E2 -8366.438} C_VEL
LIN {X 0,Y 452.496,Z 404.755,A -85,B 0,C 180,E1 -8367.329,E2 -8367.329} C_VEL
LIN {X 0,Y 452.433,Z 406.371,A -85,B 0,C 180,E1 -8369.11,E2 -8369.11} C_VEL
LIN {X 0,Y 452.41,Z 406.588,A -85,B 0,C 180,E1 -8370,E2 -8370} C_VEL
LIN {X 0,Y 452.433,Z 406.372,A -85,B 0,C 180,E1 -8370.89,E2 -8370.89} C_VEL
LIN {X 0,Y 452.496,Z 404.758,A -85,B 0,C 180,E1 -8372.671,E2 -8372.671} C_VEL
LIN {X 0,Y 452.493,Z 403.349,A -85,B 0,C 180,E1 -8373.562,E2 -8373.562} C_VEL
LIN {X 0,Y 452.567,Z 400.391,A -85,B 0,C 180,E1 -8374.9,E2 -8374.9} C_VEL
LIN {X 0,Y 452.691,Z 395.513,A -85,B 0,C 180,E1 -8376.486,E2 -8376.486} C_VEL
LIN {X 0,Y 452.926,Z 389.213,A -85,B 0,C 180,E1 -8378.028,E2 -8378.028} C_VEL
LIN {X 0,Y 453.309,Z 382.273,A -85,B 0,C 180,E1 -8379.369,E2 -8379.369} C_VEL
LIN {X 0,Y 453.736,Z 373.591,A -85,B 0,C 180,E1 -8380.712,E2 -8380.712} C_VEL
LIN {X 0,Y 454.272,Z 364.699,A -85,B 0,C 180,E1 -8381.829,E2 -8381.829} C_VEL
LIN {X 0,Y 454.78,Z 354.878,A -85,B 0,C 180,E1 -8382.842,E2 -8382.842} C_VEL
LIN {X 0,Y 455.231,Z 344.272,A -85,B 0,C 180,E1 -8383.731,E2 -8383.731} C_VEL
LIN {X 0,Y 455.826,Z 332.372,A -85,B 0,C 180,E1 -8384.51,E2 -8384.51} C_VEL
LIN {X 0,Y 456.338,Z 320,A -85,B 0,C 180,E1 -8385.121,E2 -8385.121} C_VEL
LIN {X 0,Y 454.638,Z 307.793,A -85,B 0,C 180,E1 -8385.619,E2 -8385.619} C_VEL
LIN {X 0,Y 453.085,Z 298.111,A -85,B 0,C 180,E1 -8385.923,E2 -8385.923} C_VEL
LIN {X 0,Y 453.363,Z 289.387,A -85,B 0,C 180,E1 -8388.999,E2 -8388.999} C_VEL
LIN {X 0,Y 453.611,Z 281.312,A -85,B 0,C 180,E1 -8391.83,E2 -8391.83} C_VEL
LIN {X 0,Y 453.978,Z 271.947,A -85,B 0,C 180,E1 -8395.197,E2 -8395.197} C_VEL
LIN {X 0,Y 454.376,Z 263.822,A -85,B 0,C 180,E1 -8398.159,E2 -8398.159} C_VEL
LIN {X 0,Y 454.857,Z 254.12,A -85,B 0,C 180,E1 -8401.809,E2 -8401.809} C_VEL
LIN {X 0,Y 455.268,Z 246.4,A -85,B 0,C 180,E1 -8404.832,E2 -8404.832} C_VEL
LIN {X 0,Y 455.213,Z 242.101,A -85,B 0,C 180,E1 -8406.599,E2 -8406.599} C_VEL
LIN {X 0,Y 454.173,Z 235.844,A -85,B 0,C 180,E1 -8409.379,E2 -8409.379} C_VEL
LIN {X 0,Y 453.504,Z 231.999,A -85,B 0,C 180,E1 -8411.195,E2 -8411.195} C_VEL
LIN {X 0,Y 453.488,Z 232,A -85,B 0,C 180,E1 -8414.529,E2 -8414.529} C_VEL
LIN {X 0,Y 453.451,Z 231.999,A -85,B 0,C 180,E1 -8418.069,E2 -8418.069} C_VEL
LIN {X 0,Y 453.451,Z 232.003,A -85,B 0,C 180,E1 -8420.801,E2 -8420.801} C_VEL
LIN {X 0,Y 453.455,Z 232.001,A -85,B 0,C 180,E1 -8423.917,E2 -8423.917} C_VEL
LIN {X 0,Y 453.487,Z 231.997,A -85,B 0,C 180,E1 -8427.151,E2 -8427.151} C_VEL
LIN {X 0,Y 453.466,Z 232,A -85,B 0,C 180,E1 -8430.268,E2 -8430.268} C_VEL
LIN {X 0,Y 453.445,Z 231.999,A -85,B 0,C 180,E1 -8433.29,E2 -8433.29} C_VEL
LIN {X 0,Y 453.496,Z 231.997,A -85,B 0,C 180,E1 -8436.238,E2 -8436.238} C_VEL
LIN {X 0,Y 453.487,Z 231.996,A -85,B 0,C 180,E1 -8439.118,E2 -8439.118} C_VEL
LIN {X 0,Y 453.509,Z 231.995,A -85,B 0,C 180,E1 -8441.944,E2 -8441.944} C_VEL
LIN {X 0,Y 453.541,Z 231.989,A -85,B 0,C 180,E1 -8444.726,E2 -8444.726} C_VEL
LIN {X 0,Y 453.548,Z 231.987,A -85,B 0,C 180,E1 -8448.379,E2 -8448.379} C_VEL
LIN {X 0,Y 453.576,Z 231.985,A -85,B 0,C 180,E1 -8451.086,E2 -8451.086} C_VEL
LIN {X 0,Y 453.672,Z 231.974,A -85,B 0,C 180,E1 -8453.775,E2 -8453.775} C_VEL
LIN {X 0,Y 453.748,Z 231.965,A -85,B 0,C 180,E1 -8457.337,E2 -8457.337} C_VEL
LIN {X 0,Y 453.772,Z 231.961,A -85,B 0,C 180,E1 -8460,E2 -8460} C_VEL
LIN {X 0,Y 453.717,Z 231.965,A -85,B 0,C 180,E1 -8462.664,E2 -8462.664} C_VEL
LIN {X 0,Y 453.67,Z 231.973,A -85,B 0,C 180,E1 -8466.225,E2 -8466.225} C_VEL
LIN {X 0,Y 453.59,Z 231.986,A -85,B 0,C 180,E1 -8468.913,E2 -8468.913} C_VEL
LIN {X 0,Y 453.569,Z 231.987,A -85,B 0,C 180,E1 -8472.529,E2 -8472.529} C_VEL
LIN {X 0,Y 453.542,Z 231.988,A -85,B 0,C 180,E1 -8476.196,E2 -8476.196} C_VEL
LIN {X 0,Y 453.521,Z 231.993,A -85,B 0,C 180,E1 -8479.039,E2 -8479.039} C_VEL
LIN {X 0,Y 453.481,Z 231.997,A -85,B 0,C 180,E1 -8481.836,E2 -8481.836} C_VEL
LIN {X 0,Y 453.506,Z 231.995,A -85,B 0,C 180,E1 -8484.735,E2 -8484.735} C_VEL
LIN {X 0,Y 453.479,Z 231.997,A -85,B 0,C 180,E1 -8487.946,E2 -8487.946} C_VEL
LIN {X 0,Y 453.459,Z 232.001,A -85,B 0,C 180,E1 -8490.761,E2 -8490.761} C_VEL
LIN {X 0,Y 453.472,Z 231.998,A -85,B 0,C 180,E1 -8493.913,E2 -8493.913} C_VEL
LIN {X 0,Y 453.456,Z 232,A -85,B 0,C 180,E1 -8497.19,E2 -8497.19} C_VEL
LIN {X 0,Y 453.497,Z 231.998,A -85,B 0,C 180,E1 -8500.609,E2 -8500.609} C_VEL
LIN {X 0,Y 453.464,Z 232.003,A -85,B 0,C 180,E1 -8504.222,E2 -8504.222} C_VEL
LIN {X 0,Y 453.451,Z 231.998,A -85,B 0,C 180,E1 -8507.003,E2 -8507.003} C_VEL
LIN {X 0,Y 453.497,Z 231.996,A -85,B 0,C 180,E1 -8509.409,E2 -8509.409} C_VEL
LIN {X 0,Y 453.446,Z 232.001,A -85,B 0,C 180,E1 -8512.809,E2 -8512.809} C_VEL
LIN {X 0,Y 453.347,Z 232.016,A -85,B 0,C 180,E1 -8515.249,E2 -8515.249} C_VEL
LIN {X 0,Y 453.148,Z 232.041,A -85,B 0,C 180,E1 -8517.123,E2 -8517.123} C_VEL
LIN {X 0,Y 453.01,Z 232.751,A -85,B 0,C 180,E1 -8518.57,E2 -8518.57} C_VEL
LIN {X 0,Y 452.946,Z 235.389,A -85,B 0,C 180,E1 -8521.249,E2 -8521.249} C_VEL
LIN {X 0,Y 452.876,Z 238.337,A -85,B 0,C 180,E1 -8524.245,E2 -8524.245} C_VEL
LIN {X 0,Y 452.785,Z 241.272,A -85,B 0,C 180,E1 -8527.167,E2 -8527.167} C_VEL
LIN {X 0,Y 452.738,Z 244.323,A -85,B 0,C 180,E1 -8530.031,E2 -8530.031} C_VEL
LIN {X 0,Y 452.74,Z 247.514,A -85,B 0,C 180,E1 -8532.846,E2 -8532.846} C_VEL
LIN {X 0,Y 452.778,Z 249.094,A -85,B 0,C 180,E1 -8534.188,E2 -8534.188} C_VEL
LIN {X 0,Y 456.17,Z 263.343,A -85,B 0,C 180,E1 -8534.77,E2 -8534.77} C_VEL
LIN {X 0,Y 456.716,Z 267.155,A -85,B 0,C 180,E1 -8534.949,E2 -8534.949} C_VEL
LIN {X 0,Y 456.274,Z 278.387,A -85,B 0,C 180,E1 -8535.505,E2 -8535.505} C_VEL
LIN {X 0,Y 455.907,Z 289.272,A -85,B 0,C 180,E1 -8536.21,E2 -8536.21} C_VEL
LIN {X 0,Y 455.412,Z 299.835,A -85,B 0,C 180,E1 -8537.069,E2 -8537.069} C_VEL
LIN {X 0,Y 455.236,Z 302.818,A -85,B 0,C 180,E1 -8537.352,E2 -8537.352} C_VEL
LIN {X 0,Y 454.381,Z 307.466,A -85,B 0,C 180,E1 -8537.801,E2 -8537.801} C_VEL
LIN {X 0,Y 451.111,Z 314.765,A -85,B 0,C 180,E1 -8538.548,E2 -8538.548} C_VEL
LIN {X 0,Y 447.843,Z 321.522,A -85,B 0,C 180,E1 -8539.376,E2 -8539.376} C_VEL
LIN {X 0,Y 447,Z 325.304,A -85,B 0,C 180,E1 -8539.946,E2 -8539.946} C_VEL
LIN {X 0,Y 446.535,Z 332.155,A -85,B 0,C 180,E1 -8541.173,E2 -8541.173} C_VEL
LIN {X 0,Y 446.151,Z 339.175,A -85,B 0,C 180,E1 -8542.76,E2 -8542.76} C_VEL
LIN {X 0,Y 445.84,Z 343.855,A -85,B 0,C 180,E1 -8544.119,E2 -8544.119} C_VEL
LIN {X 0,Y 445.786,Z 347.426,A -85,B 0,C 180,E1 -8545.479,E2 -8545.479} C_VEL
LIN {X 0,Y 445.697,Z 349.276,A -85,B 0,C 180,E1 -8546.384,E2 -8546.384} C_VEL
LIN {X 0,Y 445.629,Z 350.669,A -85,B 0,C 180,E1 -8547.288,E2 -8547.288} C_VEL
LIN {X 0,Y 445.44,Z 352.277,A -85,B 0,C 180,E1 -8549.096,E2 -8549.096} C_VEL
LIN {X 0,Y 445.417,Z 352.512,A -85,B 0,C 180,E1 -8550,E2 -8550} C_VEL
LIN {X 0,Y 445.527,Z 351.742,A -85,B 0,C 180,E1 -8551.808,E2 -8551.808} C_VEL
LIN {X 0,Y 445.696,Z 349.434,A -85,B 0,C 180,E1 -8553.616,E2 -8553.616} C_VEL
LIN {X 0,Y 445.771,Z 346.593,A -85,B 0,C 180,E1 -8554.974,E2 -8554.974} C_VEL
LIN {X 0,Y 445.978,Z 342.734,A -85,B 0,C 180,E1 -8556.333,E2 -8556.333} C_VEL
LIN {X 0,Y 446.192,Z 337.756,A -85,B 0,C 180,E1 -8557.694,E2 -8557.694} C_VEL
LIN {X 0,Y 446.6,Z 331.481,A -85,B 0,C 180,E1 -8559.054,E2 -8559.054} C_VEL
LIN {X 0,Y 447.079,Z 323.622,A -85,B 0,C 180,E1 -8560.415,E2 -8560.415} C_VEL
LIN {X 0,Y 447.635,Z 315.601,A -85,B 0,C 180,E1 -8561.547,E2 -8561.547} C_VEL
LIN {X 0,Y 448.178,Z 305.814,A -85,B 0,C 180,E1 -8562.682,E2 -8562.682} C_VEL
LIN {X 0,Y 448.733,Z 295.211,A -85,B 0,C 180,E1 -8563.669,E2 -8563.669} C_VEL
LIN {X 0,Y 449.285,Z 283.993,A -85,B 0,C 180,E1 -8564.494,E2 -8564.494} C_VEL
LIN {X 0,Y 449.734,Z 272.052,A -85,B 0,C 180,E1 -8565.174,E2 -8565.174} C_VEL
LIN {X 0,Y 449.825,Z 267.103,A -85,B 0,C 180,E1 -8565.403,E2 -8565.403} C_VEL
LIN {X 0,Y 447.123,Z 254.923,A -85,B 0,C 180,E1 -8565.955,E2 -8565.955} C_VEL
LIN {X 0,Y 445.71,Z 249.461,A -85,B 0,C 180,E1 -8566.158,E2 -8566.158} C_VEL
LIN {X 0,Y 445.694,Z 245.848,A -85,B 0,C 180,E1 -8569.338,E2 -8569.338} C_VEL
LIN {X 0,Y 445.712,Z 242.736,A -85,B 0,C 180,E1 -8572.237,E2 -8572.237} C_VEL
LIN {X 0,Y 445.795,Z 239.726,A -85,B 0,C 180,E1 -8575.192,E2 -8575.192} C_VEL
LIN {X 0,Y 445.871,Z 236.713,A -85,B 0,C 180,E1 -8578.221,E2 -8578.221} C_VEL
LIN {X 0,Y 445.969,Z 233.729,A -85,B 0,C 180,E1 -8581.335,E2 -8581.335} C_VEL
LIN {X 0,Y 446.008,Z 232.931,A -85,B 0,C 180,E1 -8582.395,E2 -8582.395} C_VEL
LIN {X 0,Y 446.339,Z 232.887,A -85,B 0,C 180,E1 -8585.634,E2 -8585.634} C_VEL
LIN {X 0,Y 446.427,Z 232.875,A -85,B 0,C 180,E1 -8589.029,E2 -8589.029} C_VEL
LIN {X 0,Y 446.423,Z 232.879,A -85,B 0,C 180,E1 -8592.275,E2 -8592.275} C_VEL
LIN {X 0,Y 446.452,Z 232.87,A -85,B 0,C 180,E1 -8595.104,E2 -8595.104} C_VEL
LIN {X 0,Y 446.42,Z 232.876,A -85,B 0,C 180,E1 -8598.608,E2 -8598.608} C_VEL
LIN {X 0,Y 446.426,Z 232.876,A -85,B 0,C 180,E1 -8600.971,E2 -8600.971} C_VEL
LIN {X 0,Y 446.42,Z 232.876,A -85,B 0,C 180,E1 -8604.374,E2 -8604.374} C_VEL
LIN {X 0,Y 446.422,Z 232.88,A -85,B 0,C 180,E1 -8607.638,E2 -8607.638} C_VEL
LIN {X 0,Y 446.426,Z 232.875,A -85,B 0,C 180,E1 -8610.789,E2 -8610.789} C_VEL
LIN {X 0,Y 446.44,Z 232.875,A -85,B 0,C 180,E1 -8613.846,E2 -8613.846} C_VEL
LIN {X 0,Y 446.429,Z 232.877,A -85,B 0,C 180,E1 -8616.823,E2 -8616.823} C_VEL
LIN {X 0,Y 446.446,Z 232.874,A -85,B 0,C 180,E1 -8619.737,E2 -8619.737} C_VEL
LIN {X 0,Y 446.452,Z 232.871,A -85,B 0,C 180,E1 -8622.597,E2 -8622.597} C_VEL
LIN {X 0,Y 446.465,Z 232.871,A -85,B 0,C 180,E1 -8625.412,E2 -8625.412} C_VEL
LIN {X 0,Y 446.521,Z 232.864,A -85,B 0,C 180,E1 -8628.193,E2 -8628.193} C_VEL
LIN {X 0,Y 446.604,Z 232.853,A -85,B 0,C 180,E1 -8631.858,E2 -8631.858} C_VEL
LIN {X 0,Y 446.64,Z 232.85,A -85,B 0,C 180,E1 -8634.582,E2 -8634.582} C_VEL
LIN {X 0,Y 446.662,Z 232.846,A -85,B 0,C 180,E1 -8638.197,E2 -8638.197} C_VEL
LIN {X 0,Y 446.74,Z 232.837,A -85,B 0,C 180,E1 -8640,E2 -8640} C_VEL
LIN {X 0,Y 446.694,Z 232.844,A -85,B 0,C 180,E1 -8642.705,E2 -8642.705} C_VEL
LIN {X 0,Y 446.639,Z 232.851,A -85,B 0,C 180,E1 -8646.324,E2 -8646.324} C_VEL
LIN {X 0,Y 446.53,Z 232.862,A -85,B 0,C 180,E1 -8649.056,E2 -8649.056} C_VEL
LIN {X 0,Y 446.524,Z 232.863,A -85,B 0,C 180,E1 -8652.73,E2 -8652.73} C_VEL
LIN {X 0,Y 446.493,Z 232.868,A -85,B 0,C 180,E1 -8656.459,E2 -8656.459} C_VEL
LIN {X 0,Y 446.472,Z 232.871,A -85,B 0,C 180,E1 -8659.303,E2 -8659.303} C_VEL
LIN {X 0,Y 446.421,Z 232.879,A -85,B 0,C 180,E1 -8662.2,E2 -8662.2} C_VEL
LIN {X 0,Y 446.423,Z 232.875,A -85,B 0,C 180,E1 -8665.154,E2 -8665.154} C_VEL
LIN {X 0,Y 446.438,Z 232.874,A -85,B 0,C 180,E1 -8668.182,E2 -8668.182} C_VEL
LIN {X 0,Y 446.417,Z 232.88,A -85,B 0,C 180,E1 -8671.3,E2 -8671.3} C_VEL
LIN {X 0,Y 446.43,Z 232.875,A -85,B 0,C 180,E1 -8674.523,E2 -8674.523} C_VEL
LIN {X 0,Y 446.412,Z 232.877,A -85,B 0,C 180,E1 -8678.078,E2 -8678.078} C_VEL
LIN {X 0,Y 446.408,Z 232.88,A -85,B 0,C 180,E1 -8681.394,E2 -8681.394} C_VEL
LIN {X 0,Y 446.453,Z 232.873,A -85,B 0,C 180,E1 -8685.104,E2 -8685.104} C_VEL
LIN {X 0,Y 446.457,Z 232.977,A -85,B 0,C 180,E1 -8688.537,E2 -8688.537} C_VEL
LIN {X 0,Y 447.411,Z 238.329,A -85,B 0,C 180,E1 -8691.073,E2 -8691.073} C_VEL
LIN {X 0,Y 448.286,Z 243.606,A -85,B 0,C 180,E1 -8693.434,E2 -8693.434} C_VEL
LIN {X 0,Y 448.236,Z 248.888,A -85,B 0,C 180,E1 -8695.636,E2 -8695.636} C_VEL
LIN {X 0,Y 447.764,Z 256.918,A -85,B 0,C 180,E1 -8698.804,E2 -8698.804} C_VEL
LIN {X 0,Y 447.264,Z 266.37,A -85,B 0,C 180,E1 -8702.384,E2 -8702.384} C_VEL
LIN {X 0,Y 446.896,Z 274.427,A -85,B 0,C 180,E1 -8705.371,E2 -8705.371} C_VEL
LIN {X 0,Y 446.512,Z 283.768,A -85,B 0,C 180,E1 -8708.776,E2 -8708.776} C_VEL
LIN {X 0,Y 446.221,Z 291.769,A -85,B 0,C 180,E1 -8711.639,E2 -8711.639} C_VEL
LIN {X 0,Y 446.018,Z 298.117,A -85,B 0,C 180,E1 -8713.845,E2 -8713.845} C_VEL
LIN {X 0,Y 448.164,Z 311.034,A -85,B 0,C 180,E1 -8714.265,E2 -8714.265} C_VEL
LIN {X 0,Y 449.412,Z 320.891,A -85,B 0,C 180,E1 -8714.699,E2 -8714.699} C_VEL
LIN {X 0,Y 448.946,Z 331.952,A -85,B 0,C 180,E1 -8715.263,E2 -8715.263} C_VEL
LIN {X 0,Y 448.342,Z 343.845,A -85,B 0,C 180,E1 -8716.054,E2 -8716.054} C_VEL
LIN {X 0,Y 447.739,Z 355.121,A -85,B 0,C 180,E1 -8717.019,E2 -8717.019} C_VEL
LIN {X 0,Y 447.294,Z 364.272,A -85,B 0,C 180,E1 -8717.984,E2 -8717.984} C_VEL
LIN {X 0,Y 446.715,Z 373.162,A -85,B 0,C 180,E1 -8719.118,E2 -8719.118} C_VEL
LIN {X 0,Y 446.259,Z 381.844,A -85,B 0,C 180,E1 -8720.482,E2 -8720.482} C_VEL
LIN {X 0,Y 445.884,Z 388.786,A -85,B 0,C 180,E1 -8721.845,E2 -8721.845} C_VEL
LIN {X 0,Y 445.649,Z 394.356,A -85,B 0,C 180,E1 -8723.208,E2 -8723.208} C_VEL
LIN {X 0,Y 445.541,Z 398.728,A -85,B 0,C 180,E1 -8724.569,E2 -8724.569} C_VEL
LIN {X 0,Y 445.427,Z 401.04,A -85,B 0,C 180,E1 -8725.475,E2 -8725.475} C_VEL
LIN {X 0,Y 445.397,Z 402.918,A -85,B 0,C 180,E1 -8726.381,E2 -8726.381} C_VEL
LIN {X 0,Y 445.423,Z 404.329,A -85,B 0,C 180,E1 -8727.287,E2 -8727.287} C_VEL
LIN {X 0,Y 445.372,Z 405.946,A -85,B 0,C 180,E1 -8729.096,E2 -8729.096} C_VEL
LIN {X 0,Y 445.349,Z 406.163,A -85,B 0,C 180,E1 -8730,E2 -8730} C_VEL
LIN {X 0,Y 445.372,Z 405.946,A -85,B 0,C 180,E1 -8730.904,E2 -8730.904} C_VEL
LIN {X 0,Y 445.423,Z 404.332,A -85,B 0,C 180,E1 -8732.713,E2 -8732.713} C_VEL
LIN {X 0,Y 445.397,Z 402.921,A -85,B 0,C 180,E1 -8733.619,E2 -8733.619} C_VEL
LIN {X 0,Y 445.5,Z 399.964,A -85,B 0,C 180,E1 -8734.978,E2 -8734.978} C_VEL
LIN {X 0,Y 445.587,Z 395.58,A -85,B 0,C 180,E1 -8736.451,E2 -8736.451} C_VEL
LIN {X 0,Y 445.805,Z 389.802,A -85,B 0,C 180,E1 -8737.929,E2 -8737.929} C_VEL
LIN {X 0,Y 446.186,Z 383.086,A -85,B 0,C 180,E1 -8739.291,E2 -8739.291} C_VEL
LIN {X 0,Y 446.634,Z 374.756,A -85,B 0,C 180,E1 -8740.655,E2 -8740.655} C_VEL
LIN {X 0,Y 447.17,Z 366.228,A -85,B 0,C 180,E1 -8741.79,E2 -8741.79} C_VEL
LIN {X 0,Y 447.702,Z 356.476,A -85,B 0,C 180,E1 -8742.85,E2 -8742.85} C_VEL
LIN {X 0,Y 448.241,Z 345.277,A -85,B 0,C 180,E1 -8743.834,E2 -8743.834} C_VEL
LIN {X 0,Y 448.855,Z 333.873,A -85,B 0,C 180,E1 -8744.624,E2 -8744.624} C_VEL
LIN {X 0,Y 449.373,Z 322.18,A -85,B 0,C 180,E1 -8745.245,E2 -8745.245} C_VEL
LIN {X 0,Y 449.007,Z 316.769,A -85,B 0,C 180,E1 -8745.493,E2 -8745.493} C_VEL
LIN {X 0,Y 446.839,Z 303.27,A -85,B 0,C 180,E1 -8746.009,E2 -8746.009} C_VEL
LIN {X 0,Y 446.005,Z 297.737,A -85,B 0,C 180,E1 -8746.182,E2 -8746.182} C_VEL
LIN {X 0,Y 446.326,Z 289.055,A -85,B 0,C 180,E1 -8749.31,E2 -8749.31} C_VEL
LIN {X 0,Y 446.644,Z 279.758,A -85,B 0,C 180,E1 -8752.676,E2 -8752.676} C_VEL
LIN {X 0,Y 447.083,Z 270.36,A -85,B 0,C 180,E1 -8756.114,E2 -8756.114} C_VEL
LIN {X 0,Y 447.422,Z 262.256,A -85,B 0,C 180,E1 -8759.14,E2 -8759.14} C_VEL
LIN {X 0,Y 447.918,Z 254.201,A -85,B 0,C 180,E1 -8762.241,E2 -8762.241} C_VEL
LIN {X 0,Y 448.369,Z 246.206,A -85,B 0,C 180,E1 -8765.448,E2 -8765.448} C_VEL
LIN {X 0,Y 448.184,Z 242.81,A -85,B 0,C 180,E1 -8766.895,E2 -8766.895} C_VEL
LIN {X 0,Y 446.986,Z 235.707,A -85,B 0,C 180,E1 -8770.14,E2 -8770.14} C_VEL
LIN {X 0,Y 446.455,Z 232.879,A -85,B 0,C 180,E1 -8771.539,E2 -8771.539} C_VEL
LIN {X 0,Y 446.453,Z 232.878,A -85,B 0,C 180,E1 -8775.104,E2 -8775.104} C_VEL
LIN {X 0,Y 446.409,Z 232.88,A -85,B 0,C 180,E1 -8778.607,E2 -8778.607} C_VEL
LIN {X 0,Y 446.413,Z 232.876,A -85,B 0,C 180,E1 -8781.922,E2 -8781.922} C_VEL
LIN {X 0,Y 446.432,Z 232.875,A -85,B 0,C 180,E1 -8785.477,E2 -8785.477} C_VEL
LIN {X 0,Y 446.419,Z 232.88,A -85,B 0,C 180,E1 -8788.7,E2 -8788.7} C_VEL
LIN {X 0,Y 446.427,Z 232.875,A -85,B 0,C 180,E1 -8791.836,E2 -8791.836} C_VEL
LIN {X 0,Y 446.425,Z 232.875,A -85,B 0,C 180,E1 -8794.846,E2 -8794.846} C_VEL
LIN {X 0,Y 446.453,Z 232.874,A -85,B 0,C 180,E1 -8798.245,E2 -8798.245} C_VEL
LIN {X 0,Y 446.457,Z 232.874,A -85,B 0,C 180,E1 -8801.649,E2 -8801.649} C_VEL
LIN {X 0,Y 446.51,Z 232.866,A -85,B 0,C 180,E1 -8804.48,E2 -8804.48} C_VEL
LIN {X 0,Y 446.51,Z 232.865,A -85,B 0,C 180,E1 -8808.193,E2 -8808.193} C_VEL
LIN {X 0,Y 446.523,Z 232.862,A -85,B 0,C 180,E1 -8810.944,E2 -8810.944} C_VEL
LIN {X 0,Y 446.64,Z 232.851,A -85,B 0,C 180,E1 -8813.676,E2 -8813.676} C_VEL
LIN {X 0,Y 446.695,Z 232.843,A -85,B 0,C 180,E1 -8817.295,E2 -8817.295} C_VEL
LIN {X 0,Y 446.722,Z 232.839,A -85,B 0,C 180,E1 -8820,E2 -8820} C_VEL
LIN {X 0,Y 446.667,Z 232.844,A -85,B 0,C 180,E1 -8822.706,E2 -8822.706} C_VEL
LIN {X 0,Y 446.639,Z 232.848,A -85,B 0,C 180,E1 -8826.324,E2 -8826.324} C_VEL
LIN {X 0,Y 446.538,Z 232.864,A -85,B 0,C 180,E1 -8829.055,E2 -8829.055} C_VEL
LIN {X 0,Y 446.526,Z 232.864,A -85,B 0,C 180,E1 -8832.73,E2 -8832.73} C_VEL
LIN {X 0,Y 446.489,Z 232.867,A -85,B 0,C 180,E1 -8836.459,E2 -8836.459} C_VEL
LIN {X 0,Y 446.472,Z 232.87,A -85,B 0,C 180,E1 -8839.303,E2 -8839.303} C_VEL
LIN {X 0,Y 446.423,Z 232.877,A -85,B 0,C 180,E1 -8842.199,E2 -8842.199} C_VEL
LIN {X 0,Y 446.448,Z 232.875,A -85,B 0,C 180,E1 -8845.153,E2 -8845.153} C_VEL
LIN {X 0,Y 446.441,Z 232.874,A -85,B 0,C 180,E1 -8848.182,E2 -8848.182} C_VEL
LIN {X 0,Y 446.412,Z 232.875,A -85,B 0,C 180,E1 -8851.301,E2 -8851.301} C_VEL
LIN {X 0,Y 446.427,Z 232.877,A -85,B 0,C 180,E1 -8854.523,E2 -8854.523} C_VEL
LIN {X 0,Y 446.417,Z 232.879,A -85,B 0,C 180,E1 -8858.079,E2 -8858.079} C_VEL
LIN {X 0,Y 446.426,Z 232.876,A -85,B 0,C 180,E1 -8860.917,E2 -8860.917} C_VEL
LIN {X 0,Y 446.402,Z 232.88,A -85,B 0,C 180,E1 -8863.846,E2 -8863.846} C_VEL
LIN {X 0,Y 446.401,Z 232.879,A -85,B 0,C 180,E1 -8866.403,E2 -8866.403} C_VEL
LIN {X 0,Y 446.439,Z 232.877,A -85,B 0,C 180,E1 -8869.801,E2 -8869.801} C_VEL
LIN {X 0,Y 446.39,Z 232.881,A -85,B 0,C 180,E1 -8873.253,E2 -8873.253} C_VEL
LIN {X 0,Y 446.263,Z 232.899,A -85,B 0,C 180,E1 -8875.462,E2 -8875.462} C_VEL
LIN {X 0,Y 446.009,Z 232.931,A -85,B 0,C 180,E1 -8877.604,E2 -8877.604} C_VEL
LIN {X 0,Y 445.963,Z 233.628,A -85,B 0,C 180,E1 -8878.664,E2 -8878.664} C_VEL
LIN {X 0,Y 445.874,Z 236.843,A -85,B 0,C 180,E1 -8881.969,E2 -8881.969} C_VEL
LIN {X 0,Y 445.795,Z 239.636,A -85,B 0,C 180,E1 -8884.807,E2 -8884.807} C_VEL
LIN {X 0,Y 445.717,Z 242.634,A -85,B 0,C 180,E1 -8887.763,E2 -8887.763} C_VEL
LIN {X 0,Y 445.707,Z 246.221,A -85,B 0,C 180,E1 -8891.102,E2 -8891.102} C_VEL
LIN {X 0,Y 445.731,Z 249.51,A -85,B 0,C 180,E1 -8893.935,E2 -8893.935} C_VEL
LIN {X 0,Y 449.186,Z 263.889,A -85,B 0,C 180,E1 -8894.531,E2 -8894.531} C_VEL
LIN {X 0,Y 449.859,Z 268.886,A -85,B 0,C 180,E1 -8894.772,E2 -8894.772} C_VEL
LIN {X 0,Y 449.359,Z 280.793,A -85,B 0,C 180,E1 -8895.392,E2 -8895.392} C_VEL
LIN {X 0,Y 448.877,Z 292.558,A -85,B 0,C 180,E1 -8896.212,E2 -8896.212} C_VEL
LIN {X 0,Y 448.294,Z 303.785,A -85,B 0,C 180,E1 -8897.206,E2 -8897.206} C_VEL
LIN {X 0,Y 447.746,Z 313.081,A -85,B 0,C 180,E1 -8898.226,E2 -8898.226} C_VEL
LIN {X 0,Y 447.243,Z 321.548,A -85,B 0,C 180,E1 -8899.36,E2 -8899.36} C_VEL
LIN {X 0,Y 447,Z 325.304,A -85,B 0,C 180,E1 -8899.946,E2 -8899.946} C_VEL
LIN {X 0,Y 446.172,Z 328.906,A -85,B 0,C 180,E1 -8900.54,E2 -8900.54} C_VEL
LIN {X 0,Y 441.553,Z 336.406,A -85,B 0,C 180,E1 -8901.928,E2 -8901.928} C_VEL
LIN {X 0,Y 439.414,Z 340.142,A -85,B 0,C 180,E1 -8902.793,E2 -8902.793} C_VEL
LIN {X 0,Y 439.057,Z 341.802,A -85,B 0,C 180,E1 -8903.254,E2 -8903.254} C_VEL
LIN {X 0,Y 438.717,Z 346.803,A -85,B 0,C 180,E1 -8904.945,E2 -8904.945} C_VEL
LIN {X 0,Y 438.637,Z 349.703,A -85,B 0,C 180,E1 -8906.325,E2 -8906.325} C_VEL
LIN {X 0,Y 438.552,Z 351.097,A -85,B 0,C 180,E1 -8907.244,E2 -8907.244} C_VEL
LIN {X 0,Y 438.379,Z 352.703,A -85,B 0,C 180,E1 -8909.081,E2 -8909.081} C_VEL
LIN {X 0,Y 438.354,Z 352.937,A -85,B 0,C 180,E1 -8910,E2 -8910} C_VEL
LIN {X 0,Y 438.455,Z 352.168,A -85,B 0,C 180,E1 -8911.837,E2 -8911.837} C_VEL
LIN {X 0,Y 438.636,Z 349.859,A -85,B 0,C 180,E1 -8913.674,E2 -8913.674} C_VEL
LIN {X 0,Y 438.704,Z 347.019,A -85,B 0,C 180,E1 -8915.055,E2 -8915.055} C_VEL
LIN {X 0,Y 438.949,Z 343.158,A -85,B 0,C 180,E1 -8916.435,E2 -8916.435} C_VEL
LIN {X 0,Y 439.184,Z 338.18,A -85,B 0,C 180,E1 -8917.818,E2 -8917.818} C_VEL
LIN {X 0,Y 439.6,Z 331.905,A -85,B 0,C 180,E1 -8919.199,E2 -8919.199} C_VEL
LIN {X 0,Y 440.116,Z 324.045,A -85,B 0,C 180,E1 -8920.582,E2 -8920.582} C_VEL
LIN {X 0,Y 440.697,Z 316.025,A -85,B 0,C 180,E1 -8921.732,E2 -8921.732} C_VEL
LIN {X 0,Y 441.286,Z 306.236,A -85,B 0,C 180,E1 -8922.883,E2 -8922.883} C_VEL
LIN {X 0,Y 441.817,Z 296.599,A -85,B 0,C 180,E1 -8923.804,E2 -8923.804} C_VEL
LIN {X 0,Y 442.367,Z 286.335,A -85,B 0,C 180,E1 -8924.597,E2 -8924.597} C_VEL
LIN {X 0,Y 442.834,Z 274.718,A -85,B 0,C 180,E1 -8925.298,E2 -8925.298} C_VEL
LIN {X 0,Y 442.87,Z 267.527,A -85,B 0,C 180,E1 -8925.651,E2 -8925.651} C_VEL
LIN {X 0,Y 440.089,Z 255.372,A -85,B 0,C 180,E1 -8926.216,E2 -8926.216} C_VEL
LIN {X 0,Y 438.671,Z 249.857,A -85,B 0,C 180,E1 -8926.436,E2 -8926.436} C_VEL
LIN {X 0,Y 438.626,Z 246.228,A -85,B 0,C 180,E1 -8929.662,E2 -8929.662} C_VEL
LIN {X 0,Y 438.651,Z 243.088,A -85,B 0,C 180,E1 -8932.614,E2 -8932.614} C_VEL
LIN {X 0,Y 438.745,Z 240.048,A -85,B 0,C 180,E1 -8935.626,E2 -8935.626} C_VEL
LIN {X 0,Y 438.803,Z 237.006,A -85,B 0,C 180,E1 -8938.717,E2 -8938.717} C_VEL
LIN {X 0,Y 438.923,Z 233.947,A -85,B 0,C 180,E1 -8941.936,E2 -8941.936} C_VEL
LIN {X 0,Y 439.301,Z 233.762,A -85,B 0,C 180,E1 -8945.323,E2 -8945.323} C_VEL
LIN {X 0,Y 439.371,Z 233.757,A -85,B 0,C 180,E1 -8948.596,E2 -8948.596} C_VEL
LIN {X 0,Y 439.383,Z 233.752,A -85,B 0,C 180,E1 -8951.256,E2 -8951.256} C_VEL
LIN {X 0,Y 439.4,Z 233.749,A -85,B 0,C 180,E1 -8954.73,E2 -8954.73} C_VEL
LIN {X 0,Y 439.386,Z 233.756,A -85,B 0,C 180,E1 -8957.794,E2 -8957.794} C_VEL
LIN {X 0,Y 439.391,Z 233.754,A -85,B 0,C 180,E1 -8960.223,E2 -8960.223} C_VEL
LIN {X 0,Y 439.376,Z 233.756,A -85,B 0,C 180,E1 -8963.713,E2 -8963.713} C_VEL
LIN {X 0,Y 439.374,Z 233.754,A -85,B 0,C 180,E1 -8967.054,E2 -8967.054} C_VEL
LIN {X 0,Y 439.374,Z 233.753,A -85,B 0,C 180,E1 -8970.273,E2 -8970.273} C_VEL
LIN {X 0,Y 439.38,Z 233.755,A -85,B 0,C 180,E1 -8973.393,E2 -8973.393} C_VEL
LIN {X 0,Y 439.386,Z 233.752,A -85,B 0,C 180,E1 -8976.429,E2 -8976.429} C_VEL
LIN {X 0,Y 439.391,Z 233.756,A -85,B 0,C 180,E1 -8979.397,E2 -8979.397} C_VEL
LIN {X 0,Y 439.402,Z 233.748,A -85,B 0,C 180,E1 -8982.308,E2 -8982.308} C_VEL
LIN {X 0,Y 439.437,Z 233.748,A -85,B 0,C 180,E1 -8985.174,E2 -8985.174} C_VEL
LIN {X 0,Y 439.487,Z 233.739,A -85,B 0,C 180,E1 -8988.001,E2 -8988.001} C_VEL
LIN {X 0,Y 439.551,Z 233.732,A -85,B 0,C 180,E1 -8991.726,E2 -8991.726} C_VEL
LIN {X 0,Y 439.616,Z 233.725,A -85,B 0,C 180,E1 -8994.496,E2 -8994.496} C_VEL
LIN {X 0,Y 439.632,Z 233.722,A -85,B 0,C 180,E1 -8998.168,E2 -8998.168} C_VEL
LIN {X 0,Y 439.601,Z 233.727,A -85,B 0,C 180,E1 -9000.916,E2 -9000.916} C_VEL
LIN {X 0,Y 439.643,Z 233.722,A -85,B 0,C 180,E1 -9002.749,E2 -9002.749} C_VEL
LIN {X 0,Y 439.609,Z 233.727,A -85,B 0,C 180,E1 -9006.425,E2 -9006.425} C_VEL
LIN {X 0,Y 439.493,Z 233.738,A -85,B 0,C 180,E1 -9009.202,E2 -9009.202} C_VEL
LIN {X 0,Y 439.468,Z 233.741,A -85,B 0,C 180,E1 -9012.938,E2 -9012.938} C_VEL
LIN {X 0,Y 439.45,Z 233.746,A -85,B 0,C 180,E1 -9016.349,E2 -9016.349} C_VEL
LIN {X 0,Y 439.405,Z 233.752,A -85,B 0,C 180,E1 -9019.626,E2 -9019.626} C_VEL
LIN {X 0,Y 439.366,Z 233.755,A -85,B 0,C 180,E1 -9022.575,E2 -9022.575} C_VEL
LIN {X 0,Y 439.368,Z 233.757,A -85,B 0,C 180,E1 -9025.587,E2 -9025.587} C_VEL
LIN {X 0,Y 439.391,Z 233.751,A -85,B 0,C 180,E1 -9028.675,E2 -9028.675} C_VEL
LIN {X 0,Y 439.372,Z 233.756,A -85,B 0,C 180,E1 -9032.03,E2 -9032.03} C_VEL
LIN {X 0,Y 439.395,Z 233.753,A -85,B 0,C 180,E1 -9035.34,E2 -9035.34} C_VEL
LIN {X 0,Y 439.363,Z 233.754,A -85,B 0,C 180,E1 -9038.597,E2 -9038.597} C_VEL
LIN {X 0,Y 439.36,Z 233.756,A -85,B 0,C 180,E1 -9042.209,E2 -9042.209} C_VEL
LIN {X 0,Y 439.401,Z 233.751,A -85,B 0,C 180,E1 -9045.271,E2 -9045.271} C_VEL
LIN {X 0,Y 439.421,Z 233.799,A -85,B 0,C 180,E1 -9048.173,E2 -9048.173} C_VEL
LIN {X 0,Y 440.619,Z 240.514,A -85,B 0,C 180,E1 -9051.404,E2 -9051.404} C_VEL
LIN {X 0,Y 441.391,Z 246.049,A -85,B 0,C 180,E1 -9053.905,E2 -9053.905} C_VEL
LIN {X 0,Y 441.087,Z 252.676,A -85,B 0,C 180,E1 -9056.653,E2 -9056.653} C_VEL
LIN {X 0,Y 440.615,Z 259.772,A -85,B 0,C 180,E1 -9059.466,E2 -9059.466} C_VEL
LIN {X 0,Y 440.23,Z 267.455,A -85,B 0,C 180,E1 -9062.421,E2 -9062.421} C_VEL
LIN {X 0,Y 439.813,Z 275.96,A -85,B 0,C 180,E1 -9065.621,E2 -9065.621} C_VEL
LIN {X 0,Y 439.418,Z 284.822,A -85,B 0,C 180,E1 -9068.908,E2 -9068.908} C_VEL
LIN {X 0,Y 439.117,Z 292.728,A -85,B 0,C 180,E1 -9071.815,E2 -9071.815} C_VEL
LIN {X 0,Y 438.937,Z 297.676,A -85,B 0,C 180,E1 -9073.577,E2 -9073.577} C_VEL
LIN {X 0,Y 441.099,Z 310.967,A -85,B 0,C 180,E1 -9074.019,E2 -9074.019} C_VEL
LIN {X 0,Y 442.497,Z 321.767,A -85,B 0,C 180,E1 -9074.513,E2 -9074.513} C_VEL
LIN {X 0,Y 441.957,Z 333.449,A -85,B 0,C 180,E1 -9075.142,E2 -9075.142} C_VEL
LIN {X 0,Y 441.331,Z 344.848,A -85,B 0,C 180,E1 -9075.945,E2 -9075.945} C_VEL
LIN {X 0,Y 440.71,Z 355.701,A -85,B 0,C 180,E1 -9076.909,E2 -9076.909} C_VEL
LIN {X 0,Y 440.196,Z 365.801,A -85,B 0,C 180,E1 -9078.021,E2 -9078.021} C_VEL
LIN {X 0,Y 439.621,Z 374.328,A -85,B 0,C 180,E1 -9079.173,E2 -9079.173} C_VEL
LIN {X 0,Y 439.152,Z 382.658,A -85,B 0,C 180,E1 -9080.559,E2 -9080.559} C_VEL
LIN {X 0,Y 438.751,Z 389.374,A -85,B 0,C 180,E1 -9081.943,E2 -9081.943} C_VEL
LIN {X 0,Y 438.525,Z 395.532,A -85,B 0,C 180,E1 -9083.559,E2 -9083.559} C_VEL
LIN {X 0,Y 438.434,Z 399.536,A -85,B 0,C 180,E1 -9084.942,E2 -9084.942} C_VEL
LIN {X 0,Y 438.303,Z 402.49,A -85,B 0,C 180,E1 -9086.323,E2 -9086.323} C_VEL
LIN {X 0,Y 438.351,Z 403.903,A -85,B 0,C 180,E1 -9087.243,E2 -9087.243} C_VEL
LIN {X 0,Y 438.283,Z 405.519,A -85,B 0,C 180,E1 -9089.081,E2 -9089.081} C_VEL
LIN {X 0,Y 438.29,Z 405.738,A -85,B 0,C 180,E1 -9090,E2 -9090} C_VEL
LIN {X 0,Y 438.283,Z 405.519,A -85,B 0,C 180,E1 -9090.919,E2 -9090.919} C_VEL
LIN {X 0,Y 438.351,Z 403.905,A -85,B 0,C 180,E1 -9092.757,E2 -9092.757} C_VEL
LIN {X 0,Y 438.303,Z 402.493,A -85,B 0,C 180,E1 -9093.678,E2 -9093.678} C_VEL
LIN {X 0,Y 438.435,Z 399.536,A -85,B 0,C 180,E1 -9095.058,E2 -9095.058} C_VEL
LIN {X 0,Y 438.506,Z 395.528,A -85,B 0,C 180,E1 -9096.442,E2 -9096.442} C_VEL
LIN {X 0,Y 438.753,Z 389.373,A -85,B 0,C 180,E1 -9098.057,E2 -9098.057} C_VEL
LIN {X 0,Y 439.151,Z 382.657,A -85,B 0,C 180,E1 -9099.441,E2 -9099.441} C_VEL
LIN {X 0,Y 439.621,Z 374.327,A -85,B 0,C 180,E1 -9100.827,E2 -9100.827} C_VEL
LIN {X 0,Y 440.191,Z 365.799,A -85,B 0,C 180,E1 -9101.979,E2 -9101.979} C_VEL
LIN {X 0,Y 440.73,Z 356.27,A -85,B 0,C 180,E1 -9103.035,E2 -9103.035} C_VEL
LIN {X 0,Y 441.299,Z 344.846,A -85,B 0,C 180,E1 -9104.056,E2 -9104.056} C_VEL
LIN {X 0,Y 441.959,Z 333.443,A -85,B 0,C 180,E1 -9104.858,E2 -9104.858} C_VEL
LIN {X 0,Y 442.505,Z 321.751,A -85,B 0,C 180,E1 -9105.487,E2 -9105.487} C_VEL
LIN {X 0,Y 440.974,Z 310.31,A -85,B 0,C 180,E1 -9106.007,E2 -9106.007} C_VEL
LIN {X 0,Y 438.92,Z 297.387,A -85,B 0,C 180,E1 -9106.453,E2 -9106.453} C_VEL
LIN {X 0,Y 439.257,Z 288.748,A -85,B 0,C 180,E1 -9109.633,E2 -9109.633} C_VEL
LIN {X 0,Y 439.637,Z 279.515,A -85,B 0,C 180,E1 -9113.058,E2 -9113.058} C_VEL
LIN {X 0,Y 440.086,Z 270.091,A -85,B 0,C 180,E1 -9116.561,E2 -9116.561} C_VEL
LIN {X 0,Y 440.387,Z 263.35,A -85,B 0,C 180,E1 -9119.126,E2 -9119.126} C_VEL
LIN {X 0,Y 440.919,Z 255.125,A -85,B 0,C 180,E1 -9122.35,E2 -9122.35} C_VEL
LIN {X 0,Y 441.33,Z 248.674,A -85,B 0,C 180,E1 -9124.98,E2 -9124.98} C_VEL
LIN {X 0,Y 441.281,Z 244.777,A -85,B 0,C 180,E1 -9126.641,E2 -9126.641} C_VEL
LIN {X 0,Y 440.406,Z 239.435,A -85,B 0,C 180,E1 -9129.088,E2 -9129.088} C_VEL
LIN {X 0,Y 439.412,Z 233.756,A -85,B 0,C 180,E1 -9131.891,E2 -9131.891} C_VEL
LIN {X 0,Y 439.401,Z 233.758,A -85,B 0,C 180,E1 -9135.271,E2 -9135.271} C_VEL
LIN {X 0,Y 439.36,Z 233.757,A -85,B 0,C 180,E1 -9139.017,E2 -9139.017} C_VEL
LIN {X 0,Y 439.348,Z 233.76,A -85,B 0,C 180,E1 -9142.565,E2 -9142.565} C_VEL
LIN {X 0,Y 439.402,Z 233.752,A -85,B 0,C 180,E1 -9144.844,E2 -9144.844} C_VEL
LIN {X 0,Y 439.376,Z 233.755,A -85,B 0,C 180,E1 -9148.14,E2 -9148.14} C_VEL
LIN {X 0,Y 439.403,Z 233.75,A -85,B 0,C 180,E1 -9151.606,E2 -9151.606} C_VEL
LIN {X 0,Y 439.37,Z 233.757,A -85,B 0,C 180,E1 -9154.413,E2 -9154.413} C_VEL
LIN {X 0,Y 439.367,Z 233.754,A -85,B 0,C 180,E1 -9157.425,E2 -9157.425} C_VEL
LIN {X 0,Y 439.445,Z 233.746,A -85,B 0,C 180,E1 -9160.663,E2 -9160.663} C_VEL
LIN {X 0,Y 439.466,Z 233.746,A -85,B 0,C 180,E1 -9164.225,E2 -9164.225} C_VEL
LIN {X 0,Y 439.48,Z 233.743,A -85,B 0,C 180,E1 -9168.001,E2 -9168.001} C_VEL
LIN {X 0,Y 439.505,Z 233.74,A -85,B 0,C 180,E1 -9171.725,E2 -9171.725} C_VEL
LIN {X 0,Y 439.621,Z 233.723,A -85,B 0,C 180,E1 -9174.496,E2 -9174.496} C_VEL
LIN {X 0,Y 439.637,Z 233.721,A -85,B 0,C 180,E1 -9178.168,E2 -9178.168} C_VEL
LIN {X 0,Y 439.673,Z 233.717,A -85,B 0,C 180,E1 -9180,E2 -9180} C_VEL
LIN {X 0,Y 439.619,Z 233.722,A -85,B 0,C 180,E1 -9182.749,E2 -9182.749} C_VEL
LIN {X 0,Y 439.609,Z 233.724,A -85,B 0,C 180,E1 -9186.425,E2 -9186.425} C_VEL
LIN {X 0,Y 439.501,Z 233.74,A -85,B 0,C 180,E1 -9189.202,E2 -9189.202} C_VEL
LIN {X 0,Y 439.47,Z 233.744,A -85,B 0,C 180,E1 -9192.938,E2 -9192.938} C_VEL
LIN {X 0,Y 439.449,Z 233.744,A -85,B 0,C 180,E1 -9196.347,E2 -9196.347} C_VEL
LIN {X 0,Y 439.406,Z 233.749,A -85,B 0,C 180,E1 -9199.626,E2 -9199.626} C_VEL
LIN {X 0,Y 439.369,Z 233.757,A -85,B 0,C 180,E1 -9202.575,E2 -9202.575} C_VEL
LIN {X 0,Y 439.385,Z 233.752,A -85,B 0,C 180,E1 -9205.586,E2 -9205.586} C_VEL
LIN {X 0,Y 439.393,Z 233.755,A -85,B 0,C 180,E1 -9208.675,E2 -9208.675} C_VEL
LIN {X 0,Y 439.372,Z 233.754,A -85,B 0,C 180,E1 -9212.03,E2 -9212.03} C_VEL
LIN {X 0,Y 439.396,Z 233.75,A -85,B 0,C 180,E1 -9215.34,E2 -9215.34} C_VEL
LIN {X 0,Y 439.373,Z 233.756,A -85,B 0,C 180,E1 -9218.596,E2 -9218.596} C_VEL
LIN {X 0,Y 439.385,Z 233.752,A -85,B 0,C 180,E1 -9221.255,E2 -9221.255} C_VEL
LIN {X 0,Y 439.402,Z 233.749,A -85,B 0,C 180,E1 -9224.729,E2 -9224.729} C_VEL
LIN {X 0,Y 439.387,Z 233.755,A -85,B 0,C 180,E1 -9227.794,E2 -9227.794} C_VEL
LIN {X 0,Y 439.392,Z 233.753,A -85,B 0,C 180,E1 -9230.223,E2 -9230.223} C_VEL
LIN {X 0,Y 439.338,Z 233.759,A -85,B 0,C 180,E1 -9233.115,E2 -9233.115} C_VEL
LIN {X 0,Y 439.17,Z 233.783,A -85,B 0,C 180,E1 -9235.937,E2 -9235.937} C_VEL
LIN {X 0,Y 438.904,Z 233.893,A -85,B 0,C 180,E1 -9238.101,E2 -9238.101} C_VEL
LIN {X 0,Y 438.802,Z 236.948,A -85,B 0,C 180,E1 -9241.282,E2 -9241.282} C_VEL
LIN {X 0,Y 438.742,Z 239.965,A -85,B 0,C 180,E1 -9244.373,E2 -9244.373} C_VEL
LIN {X 0,Y 438.655,Z 242.985,A -85,B 0,C 180,E1 -9247.386,E2 -9247.386} C_VEL
LIN {X 0,Y 438.662,Z 246.788,A -85,B 0,C 180,E1 -9250.956,E2 -9250.956} C_VEL
LIN {X 0,Y 438.659,Z 250.076,A -85,B 0,C 180,E1 -9253.679,E2 -9253.679} C_VEL
LIN {X 0,Y 441.954,Z 263.133,A -85,B 0,C 180,E1 -9254.224,E2 -9254.224} C_VEL
LIN {X 0,Y 443.04,Z 269.322,A -85,B 0,C 180,E1 -9254.532,E2 -9254.532} C_VEL
LIN {X 0,Y 442.527,Z 281.226,A -85,B 0,C 180,E1 -9255.162,E2 -9255.162} C_VEL
LIN {X 0,Y 442.072,Z 292.194,A -85,B 0,C 180,E1 -9255.929,E2 -9255.929} C_VEL
LIN {X 0,Y 441.455,Z 303.051,A -85,B 0,C 180,E1 -9256.887,E2 -9256.887} C_VEL
LIN {X 0,Y 440.805,Z 313.513,A -85,B 0,C 180,E1 -9258.038,E2 -9258.038} C_VEL
LIN {X 0,Y 440.292,Z 321.977,A -85,B 0,C 180,E1 -9259.19,E2 -9259.19} C_VEL
LIN {X 0,Y 439.728,Z 330.196,A -85,B 0,C 180,E1 -9260.571,E2 -9260.571} C_VEL
LIN {X 0,Y 439.341,Z 335.817,A -85,B 0,C 180,E1 -9261.722,E2 -9261.722} C_VEL
LIN {X 0,Y 439.057,Z 341.802,A -85,B 0,C 180,E1 -9263.254,E2 -9263.254} C_VEL
LIN {X 0,Y 438.335,Z 344.144,A -85,B 0,C 180,E1 -9263.956,E2 -9263.956} C_VEL
LIN {X 0,Y 435.291,Z 347.485,A -85,B 0,C 180,E1 -9265.114,E2 -9265.114} C_VEL
LIN {X 0,Y 432.714,Z 349.674,A -85,B 0,C 180,E1 -9266.069,E2 -9266.069} C_VEL
LIN {X 0,Y 431.587,Z 350.992,A -85,B 0,C 180,E1 -9266.821,E2 -9266.821} C_VEL
LIN {X 0,Y 431.485,Z 351.342,A -85,B 0,C 180,E1 -9267.077,E2 -9267.077} C_VEL
LIN {X 0,Y 431.372,Z 352.517,A -85,B 0,C 180,E1 -9268.133,E2 -9268.133} C_VEL
LIN {X 0,Y 431.293,Z 353.362,A -85,B 0,C 180,E1 -9270,E2 -9270} C_VEL
LIN {X 0,Y 431.32,Z 353.175,A -85,B 0,C 180,E1 -9270.934,E2 -9270.934} C_VEL
LIN {X 0,Y 431.468,Z 351.632,A -85,B 0,C 180,E1 -9272.801,E2 -9272.801} C_VEL
LIN {X 0,Y 431.578,Z 350.285,A -85,B 0,C 180,E1 -9273.735,E2 -9273.735} C_VEL
LIN {X 0,Y 431.624,Z 347.446,A -85,B 0,C 180,E1 -9275.138,E2 -9275.138} C_VEL
LIN {X 0,Y 431.91,Z 343.583,A -85,B 0,C 180,E1 -9276.54,E2 -9276.54} C_VEL
LIN {X 0,Y 432.157,Z 338.606,A -85,B 0,C 180,E1 -9277.945,E2 -9277.945} C_VEL
LIN {X 0,Y 432.615,Z 332.329,A -85,B 0,C 180,E1 -9279.349,E2 -9279.349} C_VEL
LIN {X 0,Y 433.163,Z 324.468,A -85,B 0,C 180,E1 -9280.754,E2 -9280.754} C_VEL
LIN {X 0,Y 433.764,Z 316.448,A -85,B 0,C 180,E1 -9281.922,E2 -9281.922} C_VEL
LIN {X 0,Y 434.398,Z 306.657,A -85,B 0,C 180,E1 -9283.091,E2 -9283.091} C_VEL
LIN {X 0,Y 435.022,Z 295.576,A -85,B 0,C 180,E1 -9284.149,E2 -9284.149} C_VEL
LIN {X 0,Y 435.669,Z 283.076,A -85,B 0,C 180,E1 -9285.077,E2 -9285.077} C_VEL
LIN {X 0,Y 436.157,Z 270.523,A -85,B 0,C 180,E1 -9285.778,E2 -9285.778} C_VEL
LIN {X 0,Y 435.071,Z 264.103,A -85,B 0,C 180,E1 -9286.107,E2 -9286.107} C_VEL
LIN {X 0,Y 431.764,Z 251.291,A -85,B 0,C 180,E1 -9286.663,E2 -9286.663} C_VEL
LIN {X 0,Y 431.603,Z 250.28,A -85,B 0,C 180,E1 -9286.704,E2 -9286.704} C_VEL
LIN {X 0,Y 431.563,Z 246.61,A -85,B 0,C 180,E1 -9289.998,E2 -9289.998} C_VEL
LIN {X 0,Y 431.602,Z 243.442,A -85,B 0,C 180,E1 -9293.005,E2 -9293.005} C_VEL
LIN {X 0,Y 431.71,Z 240.373,A -85,B 0,C 180,E1 -9296.075,E2 -9296.075} C_VEL
LIN {X 0,Y 431.781,Z 237.301,A -85,B 0,C 180,E1 -9299.229,E2 -9299.229} C_VEL
LIN {X 0,Y 431.88,Z 234.691,A -85,B 0,C 180,E1 -9302.199,E2 -9302.199} C_VEL
LIN {X 0,Y 432.189,Z 234.651,A -85,B 0,C 180,E1 -9304.691,E2 -9304.691} C_VEL
LIN {X 0,Y 432.333,Z 234.633,A -85,B 0,C 180,E1 -9308.15,E2 -9308.15} C_VEL
LIN {X 0,Y 432.326,Z 234.632,A -85,B 0,C 180,E1 -9311.601,E2 -9311.601} C_VEL
LIN {X 0,Y 432.335,Z 234.631,A -85,B 0,C 180,E1 -9314.347,E2 -9314.347} C_VEL
LIN {X 0,Y 432.318,Z 234.632,A -85,B 0,C 180,E1 -9317.016,E2 -9317.016} C_VEL
LIN {X 0,Y 432.334,Z 234.633,A -85,B 0,C 180,E1 -9319.821,E2 -9319.821} C_VEL
LIN {X 0,Y 432.308,Z 234.634,A -85,B 0,C 180,E1 -9323.022,E2 -9323.022} C_VEL
LIN {X 0,Y 432.36,Z 234.629,A -85,B 0,C 180,E1 -9325.997,E2 -9325.997} C_VEL
LIN {X 0,Y 432.348,Z 234.633,A -85,B 0,C 180,E1 -9329.49,E2 -9329.49} C_VEL
LIN {X 0,Y 432.341,Z 234.631,A -85,B 0,C 180,E1 -9331.874,E2 -9331.874} C_VEL
LIN {X 0,Y 432.381,Z 234.627,A -85,B 0,C 180,E1 -9335.538,E2 -9335.538} C_VEL
LIN {X 0,Y 432.353,Z 234.63,A -85,B 0,C 180,E1 -9339.046,E2 -9339.046} C_VEL
LIN {X 0,Y 432.359,Z 234.626,A -85,B 0,C 180,E1 -9342.01,E2 -9342.01} C_VEL
LIN {X 0,Y 432.384,Z 234.628,A -85,B 0,C 180,E1 -9344.926,E2 -9344.926} C_VEL
LIN {X 0,Y 432.463,Z 234.614,A -85,B 0,C 180,E1 -9347.803,E2 -9347.803} C_VEL
LIN {X 0,Y 432.495,Z 234.611,A -85,B 0,C 180,E1 -9351.59,E2 -9351.59} C_VEL
LIN {X 0,Y 432.593,Z 234.599,A -85,B 0,C 180,E1 -9354.406,E2 -9354.406} C_VEL
LIN {X 0,Y 432.601,Z 234.597,A -85,B 0,C 180,E1 -9358.138,E2 -9358.138} C_VEL
LIN {X 0,Y 432.561,Z 234.604,A -85,B 0,C 180,E1 -9360.931,E2 -9360.931} C_VEL
LIN {X 0,Y 432.595,Z 234.6,A -85,B 0,C 180,E1 -9362.794,E2 -9362.794} C_VEL
LIN {X 0,Y 432.596,Z 234.598,A -85,B 0,C 180,E1 -9365.594,E2 -9365.594} C_VEL
LIN {X 0,Y 432.465,Z 234.618,A -85,B 0,C 180,E1 -9368.41,E2 -9368.41} C_VEL
LIN {X 0,Y 432.456,Z 234.62,A -85,B 0,C 180,E1 -9372.197,E2 -9372.197} C_VEL
LIN {X 0,Y 432.433,Z 234.621,A -85,B 0,C 180,E1 -9376.039,E2 -9376.039} C_VEL
LIN {X 0,Y 432.39,Z 234.626,A -85,B 0,C 180,E1 -9379.485,E2 -9379.485} C_VEL
LIN {X 0,Y 432.314,Z 234.632,A -85,B 0,C 180,E1 -9382.965,E2 -9382.965} C_VEL
LIN {X 0,Y 432.319,Z 234.634,A -85,B 0,C 180,E1 -9386.035,E2 -9386.035} C_VEL
LIN {X 0,Y 432.328,Z 234.632,A -85,B 0,C 180,E1 -9389.189,E2 -9389.189} C_VEL
LIN {X 0,Y 432.325,Z 234.632,A -85,B 0,C 180,E1 -9392.443,E2 -9392.443} C_VEL
LIN {X 0,Y 432.345,Z 234.633,A -85,B 0,C 180,E1 -9395.632,E2 -9395.632} C_VEL
LIN {X 0,Y 432.326,Z 234.631,A -85,B 0,C 180,E1 -9398.712,E2 -9398.712} C_VEL
LIN {X 0,Y 432.31,Z 234.633,A -85,B 0,C 180,E1 -9401.8,E2 -9401.8} C_VEL
LIN {X 0,Y 432.335,Z 234.634,A -85,B 0,C 180,E1 -9404.347,E2 -9404.347} C_VEL
LIN {X 0,Y 432.372,Z 234.789,A -85,B 0,C 180,E1 -9407.894,E2 -9407.894} C_VEL
LIN {X 0,Y 433.419,Z 240.628,A -85,B 0,C 180,E1 -9410.773,E2 -9410.773} C_VEL
LIN {X 0,Y 434.325,Z 245.874,A -85,B 0,C 180,E1 -9413.222,E2 -9413.222} C_VEL
LIN {X 0,Y 434.265,Z 251.438,A -85,B 0,C 180,E1 -9415.626,E2 -9415.626} C_VEL
LIN {X 0,Y 433.738,Z 259.138,A -85,B 0,C 180,E1 -9418.768,E2 -9418.768} C_VEL
LIN {X 0,Y 433.186,Z 268.525,A -85,B 0,C 180,E1 -9422.459,E2 -9422.459} C_VEL
LIN {X 0,Y 432.687,Z 277.901,A -85,B 0,C 180,E1 -9426.042,E2 -9426.042} C_VEL
LIN {X 0,Y 432.256,Z 287.154,A -85,B 0,C 180,E1 -9429.539,E2 -9429.539} C_VEL
LIN {X 0,Y 431.948,Z 294.986,A -85,B 0,C 180,E1 -9432.482,E2 -9432.482} C_VEL
LIN {X 0,Y 431.87,Z 297.175,A -85,B 0,C 180,E1 -9433.279,E2 -9433.279} C_VEL
LIN {X 0,Y 434.299,Z 312.339,A -85,B 0,C 180,E1 -9433.829,E2 -9433.829} C_VEL
LIN {X 0,Y 435.583,Z 322.55,A -85,B 0,C 180,E1 -9434.321,E2 -9434.321} C_VEL
LIN {X 0,Y 434.963,Z 334.792,A -85,B 0,C 180,E1 -9435.018,E2 -9435.018} C_VEL
LIN {X 0,Y 434.315,Z 345.852,A -85,B 0,C 180,E1 -9435.833,E2 -9435.833} C_VEL
LIN {X 0,Y 433.71,Z 355.781,A -85,B 0,C 180,E1 -9436.745,E2 -9436.745} C_VEL
LIN {X 0,Y 433.204,Z 365.37,A -85,B 0,C 180,E1 -9437.825,E2 -9437.825} C_VEL
LIN {X 0,Y 432.588,Z 373.897,A -85,B 0,C 180,E1 -9438.995,E2 -9438.995} C_VEL
LIN {X 0,Y 432.103,Z 382.227,A -85,B 0,C 180,E1 -9440.403,E2 -9440.403} C_VEL
LIN {X 0,Y 431.711,Z 388.946,A -85,B 0,C 180,E1 -9441.811,E2 -9441.811} C_VEL
LIN {X 0,Y 431.465,Z 395.104,A -85,B 0,C 180,E1 -9443.453,E2 -9443.453} C_VEL
LIN {X 0,Y 431.369,Z 399.108,A -85,B 0,C 180,E1 -9444.859,E2 -9444.859} C_VEL
LIN {X 0,Y 431.21,Z 402.061,A -85,B 0,C 180,E1 -9446.262,E2 -9446.262} C_VEL
LIN {X 0,Y 431.28,Z 403.476,A -85,B 0,C 180,E1 -9447.198,E2 -9447.198} C_VEL
LIN {X 0,Y 431.198,Z 405.092,A -85,B 0,C 180,E1 -9449.066,E2 -9449.066} C_VEL
LIN {X 0,Y 431.216,Z 405.312,A -85,B 0,C 180,E1 -9450,E2 -9450} C_VEL
LIN {X 0,Y 431.198,Z 405.092,A -85,B 0,C 180,E1 -9450.934,E2 -9450.934} C_VEL
LIN {X 0,Y 431.28,Z 403.479,A -85,B 0,C 180,E1 -9452.802,E2 -9452.802} C_VEL
LIN {X 0,Y 431.21,Z 402.065,A -85,B 0,C 180,E1 -9453.738,E2 -9453.738} C_VEL
LIN {X 0,Y 431.369,Z 399.109,A -85,B 0,C 180,E1 -9455.141,E2 -9455.141} C_VEL
LIN {X 0,Y 431.441,Z 395.1,A -85,B 0,C 180,E1 -9456.548,E2 -9456.548} C_VEL
LIN {X 0,Y 431.712,Z 388.945,A -85,B 0,C 180,E1 -9458.19,E2 -9458.19} C_VEL
LIN {X 0,Y 432.102,Z 382.227,A -85,B 0,C 180,E1 -9459.597,E2 -9459.597} C_VEL
LIN {X 0,Y 432.588,Z 373.895,A -85,B 0,C 180,E1 -9461.005,E2 -9461.005} C_VEL
LIN {X 0,Y 433.199,Z 365.368,A -85,B 0,C 180,E1 -9462.176,E2 -9462.176} C_VEL
LIN {X 0,Y 433.81,Z 355.382,A -85,B 0,C 180,E1 -9463.293,E2 -9463.293} C_VEL
LIN {X 0,Y 434.378,Z 344.416,A -85,B 0,C 180,E1 -9464.285,E2 -9464.285} C_VEL
LIN {X 0,Y 435.104,Z 333.016,A -85,B 0,C 180,E1 -9465.098,E2 -9465.098} C_VEL
LIN {X 0,Y 435.572,Z 321.318,A -85,B 0,C 180,E1 -9465.74,E2 -9465.74} C_VEL
LIN {X 0,Y 433.632,Z 308.406,A -85,B 0,C 180,E1 -9466.333,E2 -9466.333} C_VEL
LIN {X 0,Y 431.865,Z 297.07,A -85,B 0,C 180,E1 -9466.721,E2 -9466.721} C_VEL
LIN {X 0,Y 432.209,Z 288.465,A -85,B 0,C 180,E1 -9469.967,E2 -9469.967} C_VEL
LIN {X 0,Y 432.557,Z 280.551,A -85,B 0,C 180,E1 -9472.951,E2 -9472.951} C_VEL
LIN {X 0,Y 433.031,Z 271.447,A -85,B 0,C 180,E1 -9476.396,E2 -9476.396} C_VEL
LIN {X 0,Y 433.361,Z 264.424,A -85,B 0,C 180,E1 -9479.113,E2 -9479.113} C_VEL
LIN {X 0,Y 433.895,Z 256.408,A -85,B 0,C 180,E1 -9482.311,E2 -9482.311} C_VEL
LIN {X 0,Y 434.346,Z 249.796,A -85,B 0,C 180,E1 -9485.059,E2 -9485.059} C_VEL
LIN {X 0,Y 434.304,Z 245.859,A -85,B 0,C 180,E1 -9486.78,E2 -9486.78} C_VEL
LIN {X 0,Y 433.411,Z 240.597,A -85,B 0,C 180,E1 -9489.228,E2 -9489.228} C_VEL
LIN {X 0,Y 432.38,Z 234.633,A -85,B 0,C 180,E1 -9492.184,E2 -9492.184} C_VEL
LIN {X 0,Y 432.336,Z 234.633,A -85,B 0,C 180,E1 -9495.665,E2 -9495.665} C_VEL
LIN {X 0,Y 432.314,Z 234.634,A -85,B 0,C 180,E1 -9498.401,E2 -9498.401} C_VEL
LIN {X 0,Y 432.332,Z 234.63,A -85,B 0,C 180,E1 -9501.849,E2 -9501.849} C_VEL
LIN {X 0,Y 432.343,Z 234.63,A -85,B 0,C 180,E1 -9505.323,E2 -9505.323} C_VEL
LIN {X 0,Y 432.324,Z 234.635,A -85,B 0,C 180,E1 -9508.654,E2 -9508.654} C_VEL
LIN {X 0,Y 432.331,Z 234.631,A -85,B 0,C 180,E1 -9511.873,E2 -9511.873} C_VEL
LIN {X 0,Y 432.357,Z 234.627,A -85,B 0,C 180,E1 -9515.546,E2 -9515.546} C_VEL
LIN {X 0,Y 432.355,Z 234.628,A -85,B 0,C 180,E1 -9519.046,E2 -9519.046} C_VEL
LIN {X 0,Y 432.378,Z 234.627,A -85,B 0,C 180,E1 -9522.011,E2 -9522.011} C_VEL
LIN {X 0,Y 432.396,Z 234.622,A -85,B 0,C 180,E1 -9524.926,E2 -9524.926} C_VEL
LIN {X 0,Y 432.458,Z 234.619,A -85,B 0,C 180,E1 -9527.803,E2 -9527.803} C_VEL
LIN {X 0,Y 432.465,Z 234.618,A -85,B 0,C 180,E1 -9531.59,E2 -9531.59} C_VEL
LIN {X 0,Y 432.597,Z 234.598,A -85,B 0,C 180,E1 -9534.406,E2 -9534.406} C_VEL
LIN {X 0,Y 432.607,Z 234.597,A -85,B 0,C 180,E1 -9538.138,E2 -9538.138} C_VEL
LIN {X 0,Y 432.625,Z 234.595,A -85,B 0,C 180,E1 -9540,E2 -9540} C_VEL
LIN {X 0,Y 432.572,Z 234.6,A -85,B 0,C 180,E1 -9542.794,E2 -9542.794} C_VEL
LIN {X 0,Y 432.593,Z 234.6,A -85,B 0,C 180,E1 -9545.594,E2 -9545.594} C_VEL
LIN {X 0,Y 432.469,Z 234.614,A -85,B 0,C 180,E1 -9548.41,E2 -9548.41} C_VEL
LIN {X 0,Y 432.464,Z 234.614,A -85,B 0,C 180,E1 -9552.197,E2 -9552.197} C_VEL
LIN {X 0,Y 432.425,Z 234.618,A -85,B 0,C 180,E1 -9556.039,E2 -9556.039} C_VEL
LIN {X 0,Y 432.391,Z 234.624,A -85,B 0,C 180,E1 -9559.485,E2 -9559.485} C_VEL
LIN {X 0,Y 432.322,Z 234.634,A -85,B 0,C 180,E1 -9562.964,E2 -9562.964} C_VEL
LIN {X 0,Y 432.344,Z 234.633,A -85,B 0,C 180,E1 -9565.002,E2 -9565.002} C_VEL
LIN {X 0,Y 432.343,Z 234.631,A -85,B 0,C 180,E1 -9568.126,E2 -9568.126} C_VEL
LIN {X 0,Y 432.321,Z 234.63,A -85,B 0,C 180,E1 -9571.346,E2 -9571.346} C_VEL
LIN {X 0,Y 432.341,Z 234.631,A -85,B 0,C 180,E1 -9574.677,E2 -9574.677} C_VEL
LIN {X 0,Y 432.337,Z 234.633,A -85,B 0,C 180,E1 -9578.15,E2 -9578.15} C_VEL
LIN {X 0,Y 432.328,Z 234.632,A -85,B 0,C 180,E1 -9581.601,E2 -9581.601} C_VEL
LIN {X 0,Y 432.337,Z 234.633,A -85,B 0,C 180,E1 -9584.347,E2 -9584.347} C_VEL
LIN {X 0,Y 432.32,Z 234.631,A -85,B 0,C 180,E1 -9587.016,E2 -9587.016} C_VEL
LIN {X 0,Y 432.335,Z 234.634,A -85,B 0,C 180,E1 -9589.821,E2 -9589.821} C_VEL
LIN {X 0,Y 432.298,Z 234.635,A -85,B 0,C 180,E1 -9593.021,E2 -9593.021} C_VEL
LIN {X 0,Y 432.12,Z 234.661,A -85,B 0,C 180,E1 -9596.044,E2 -9596.044} C_VEL
LIN {X 0,Y 431.886,Z 234.691,A -85,B 0,C 180,E1 -9597.8,E2 -9597.8} C_VEL
LIN {X 0,Y 431.819,Z 236.208,A -85,B 0,C 180,E1 -9599.699,E2 -9599.699} C_VEL
LIN {X 0,Y 431.719,Z 239.255,A -85,B 0,C 180,E1 -9602.882,E2 -9602.882} C_VEL
LIN {X 0,Y 431.683,Z 242.295,A -85,B 0,C 180,E1 -9605.982,E2 -9605.982} C_VEL
LIN {X 0,Y 431.565,Z 245.432,A -85,B 0,C 180,E1 -9609.006,E2 -9609.006} C_VEL
LIN {X 0,Y 431.548,Z 248.7,A -85,B 0,C 180,E1 -9611.975,E2 -9611.975} C_VEL
LIN {X 0,Y 431.614,Z 250.314,A -85,B 0,C 180,E1 -9613.376,E2 -9613.376} C_VEL
LIN {X 0,Y 435.455,Z 265.895,A -85,B 0,C 180,E1 -9614.075,E2 -9614.075} C_VEL
LIN {X 0,Y 436.196,Z 271.051,A -85,B 0,C 180,E1 -9614.343,E2 -9614.343} C_VEL
LIN {X 0,Y 435.598,Z 283.445,A -85,B 0,C 180,E1 -9615.04,E2 -9615.04} C_VEL
LIN {X 0,Y 435.097,Z 294.029,A -85,B 0,C 180,E1 -9615.817,E2 -9615.817} C_VEL
LIN {X 0,Y 434.495,Z 304.647,A -85,B 0,C 180,E1 -9616.793,E2 -9616.793} C_VEL
LIN {X 0,Y 433.869,Z 313.944,A -85,B 0,C 180,E1 -9617.843,E2 -9617.843} C_VEL
LIN {X 0,Y 433.323,Z 322.407,A -85,B 0,C 180,E1 -9619.014,E2 -9619.014} C_VEL
LIN {X 0,Y 432.742,Z 330.625,A -85,B 0,C 180,E1 -9620.417,E2 -9620.417} C_VEL
LIN {X 0,Y 432.332,Z 336.246,A -85,B 0,C 180,E1 -9621.587,E2 -9621.587} C_VEL
LIN {X 0,Y 431.975,Z 342.428,A -85,B 0,C 180,E1 -9623.203,E2 -9623.203} C_VEL
LIN {X 0,Y 431.656,Z 347.231,A -85,B 0,C 180,E1 -9624.862,E2 -9624.862} C_VEL
LIN {X 0,Y 431.58,Z 350.129,A -85,B 0,C 180,E1 -9626.265,E2 -9626.265} C_VEL
LIN {X 0,Y 431.485,Z 351.342,A -85,B 0,C 180,E1 -9627.077,E2 -9627.077} C_VEL
LIN {X 0,Y 430.77,Z 352.374,A -85,B 0,C 180,E1 -9627.844,E2 -9627.844} C_VEL
LIN {X 0,Y 427.83,Z 353.493,A -85,B 0,C 180,E1 -9629.1,E2 -9629.1} C_VEL
LIN {X 0,Y 425.37,Z 353.782,A -85,B 0,C 180,E1 -9630.118,E2 -9630.118} C_VEL
LIN {X 0,Y 424.325,Z 353.617,A -85,B 0,C 180,E1 -9630.907,E2 -9630.907} C_VEL
LIN {X 0,Y 424.246,Z 353.464,A -85,B 0,C 180,E1 -9631.173,E2 -9631.173} C_VEL
LIN {X 0,Y 424.398,Z 352.058,A -85,B 0,C 180,E1 -9632.847,E2 -9632.847} C_VEL
LIN {X 0,Y 424.521,Z 350.71,A -85,B 0,C 180,E1 -9633.797,E2 -9633.797} C_VEL
LIN {X 0,Y 424.55,Z 347.873,A -85,B 0,C 180,E1 -9635.224,E2 -9635.224} C_VEL
LIN {X 0,Y 424.874,Z 344.009,A -85,B 0,C 180,E1 -9636.649,E2 -9636.649} C_VEL
LIN {X 0,Y 425.151,Z 339.03,A -85,B 0,C 180,E1 -9638.077,E2 -9638.077} C_VEL
LIN {X 0,Y 425.613,Z 332.754,A -85,B 0,C 180,E1 -9639.505,E2 -9639.505} C_VEL
LIN {X 0,Y 426.217,Z 324.891,A -85,B 0,C 180,E1 -9640.931,E2 -9640.931} C_VEL
LIN {X 0,Y 426.822,Z 316.871,A -85,B 0,C 180,E1 -9642.119,E2 -9642.119} C_VEL
LIN {X 0,Y 427.518,Z 307.079,A -85,B 0,C 180,E1 -9643.306,E2 -9643.306} C_VEL
LIN {X 0,Y 428.094,Z 297.441,A -85,B 0,C 180,E1 -9644.256,E2 -9644.256} C_VEL
LIN {X 0,Y 428.694,Z 287.005,A -85,B 0,C 180,E1 -9645.085,E2 -9645.085} C_VEL
LIN {X 0,Y 429.218,Z 274.429,A -85,B 0,C 180,E1 -9645.857,E2 -9645.857} C_VEL
LIN {X 0,Y 429.168,Z 269.657,A -85,B 0,C 180,E1 -9646.103,E2 -9646.103} C_VEL
LIN {X 0,Y 426.305,Z 257.454,A -85,B 0,C 180,E1 -9646.713,E2 -9646.713} C_VEL
LIN {X 0,Y 424.526,Z 250.676,A -85,B 0,C 180,E1 -9647.008,E2 -9647.008} C_VEL
LIN {X 0,Y 424.498,Z 246.995,A -85,B 0,C 180,E1 -9650.345,E2 -9650.345} C_VEL
LIN {X 0,Y 424.559,Z 243.798,A -85,B 0,C 180,E1 -9653.409,E2 -9653.409} C_VEL
LIN {X 0,Y 424.647,Z 240.705,A -85,B 0,C 180,E1 -9656.542,E2 -9656.542} C_VEL
LIN {X 0,Y 424.747,Z 237.597,A -85,B 0,C 180,E1 -9659.761,E2 -9659.761} C_VEL
LIN {X 0,Y 424.797,Z 235.573,A -85,B 0,C 180,E1 -9661.966,E2 -9661.966} C_VEL
LIN {X 0,Y 425.121,Z 235.533,A -85,B 0,C 180,E1 -9664.25,E2 -9664.25} C_VEL
LIN {X 0,Y 425.274,Z 235.51,A -85,B 0,C 180,E1 -9667.51,E2 -9667.51} C_VEL
LIN {X 0,Y 425.278,Z 235.511,A -85,B 0,C 180,E1 -9670.52,E2 -9670.52} C_VEL
LIN {X 0,Y 425.263,Z 235.515,A -85,B 0,C 180,E1 -9673.956,E2 -9673.956} C_VEL
LIN {X 0,Y 425.272,Z 235.51,A -85,B 0,C 180,E1 -9677.346,E2 -9677.346} C_VEL
LIN {X 0,Y 425.286,Z 235.511,A -85,B 0,C 180,E1 -9679.872,E2 -9679.872} C_VEL
LIN {X 0,Y 425.279,Z 235.509,A -85,B 0,C 180,E1 -9682.489,E2 -9682.489} C_VEL
LIN {X 0,Y 425.308,Z 235.51,A -85,B 0,C 180,E1 -9685.817,E2 -9685.817} C_VEL
LIN {X 0,Y 425.292,Z 235.509,A -85,B 0,C 180,E1 -9689.239,E2 -9689.239} C_VEL
LIN {X 0,Y 425.268,Z 235.51,A -85,B 0,C 180,E1 -9692.436,E2 -9692.436} C_VEL
LIN {X 0,Y 425.35,Z 235.503,A -85,B 0,C 180,E1 -9695.602,E2 -9695.602} C_VEL
LIN {X 0,Y 425.296,Z 235.508,A -85,B 0,C 180,E1 -9698.682,E2 -9698.682} C_VEL
LIN {X 0,Y 425.321,Z 235.504,A -85,B 0,C 180,E1 -9701.702,E2 -9701.702} C_VEL
LIN {X 0,Y 425.338,Z 235.503,A -85,B 0,C 180,E1 -9704.67,E2 -9704.67} C_VEL
LIN {X 0,Y 425.415,Z 235.493,A -85,B 0,C 180,E1 -9707.598,E2 -9707.598} C_VEL
LIN {X 0,Y 425.446,Z 235.489,A -85,B 0,C 180,E1 -9711.45,E2 -9711.45} C_VEL
LIN {X 0,Y 425.551,Z 235.477,A -85,B 0,C 180,E1 -9714.313,E2 -9714.313} C_VEL
LIN {X 0,Y 425.57,Z 235.473,A -85,B 0,C 180,E1 -9718.107,E2 -9718.107} C_VEL
LIN {X 0,Y 425.522,Z 235.481,A -85,B 0,C 180,E1 -9720.946,E2 -9720.946} C_VEL
LIN {X 0,Y 425.548,Z 235.478,A -85,B 0,C 180,E1 -9722.84,E2 -9722.84} C_VEL
LIN {X 0,Y 425.551,Z 235.476,A -85,B 0,C 180,E1 -9725.687,E2 -9725.687} C_VEL
LIN {X 0,Y 425.409,Z 235.496,A -85,B 0,C 180,E1 -9728.551,E2 -9728.551} C_VEL
LIN {X 0,Y 425.411,Z 235.495,A -85,B 0,C 180,E1 -9732.402,E2 -9732.402} C_VEL
LIN {X 0,Y 425.391,Z 235.497,A -85,B 0,C 180,E1 -9736.312,E2 -9736.312} C_VEL
LIN {X 0,Y 425.331,Z 235.506,A -85,B 0,C 180,E1 -9739.636,E2 -9739.636} C_VEL
LIN {X 0,Y 425.289,Z 235.509,A -85,B 0,C 180,E1 -9742.339,E2 -9742.339} C_VEL
LIN {X 0,Y 425.261,Z 235.513,A -85,B 0,C 180,E1 -9745.448,E2 -9745.448} C_VEL
LIN {X 0,Y 425.309,Z 235.505,A -85,B 0,C 180,E1 -9748.86,E2 -9748.86} C_VEL
LIN {X 0,Y 425.267,Z 235.513,A -85,B 0,C 180,E1 -9751.927,E2 -9751.927} C_VEL
LIN {X 0,Y 425.301,Z 235.509,A -85,B 0,C 180,E1 -9755.336,E2 -9755.336} C_VEL
LIN {X 0,Y 425.282,Z 235.51,A -85,B 0,C 180,E1 -9758.901,E2 -9758.901} C_VEL
LIN {X 0,Y 425.262,Z 235.516,A -85,B 0,C 180,E1 -9762.655,E2 -9762.655} C_VEL
LIN {X 0,Y 425.286,Z 235.509,A -85,B 0,C 180,E1 -9765.283,E2 -9765.283} C_VEL
LIN {X 0,Y 425.346,Z 235.694,A -85,B 0,C 180,E1 -9767.56,E2 -9767.56} C_VEL
LIN {X 0,Y 426.227,Z 240.451,A -85,B 0,C 180,E1 -9769.979,E2 -9769.979} C_VEL
LIN {X 0,Y 427.315,Z 246.985,A -85,B 0,C 180,E1 -9773.108,E2 -9773.108} C_VEL
LIN {X 0,Y 427.325,Z 251.988,A -85,B 0,C 180,E1 -9775.318,E2 -9775.318} C_VEL
LIN {X 0,Y 426.836,Z 258.889,A -85,B 0,C 180,E1 -9778.204,E2 -9778.204} C_VEL
LIN {X 0,Y 426.239,Z 268.254,A -85,B 0,C 180,E1 -9781.971,E2 -9781.971} C_VEL
LIN {X 0,Y 425.697,Z 277.599,A -85,B 0,C 180,E1 -9785.623,E2 -9785.623} C_VEL
LIN {X 0,Y 425.236,Z 286.829,A -85,B 0,C 180,E1 -9789.186,E2 -9789.186} C_VEL
LIN {X 0,Y 424.894,Z 294.635,A -85,B 0,C 180,E1 -9792.182,E2 -9792.182} C_VEL
LIN {X 0,Y 424.79,Z 296.751,A -85,B 0,C 180,E1 -9792.992,E2 -9792.992} C_VEL
LIN {X 0,Y 427.195,Z 312.022,A -85,B 0,C 180,E1 -9793.558,E2 -9793.558} C_VEL
LIN {X 0,Y 428.67,Z 323.254,A -85,B 0,C 180,E1 -9794.122,E2 -9794.122} C_VEL
LIN {X 0,Y 427.97,Z 336.135,A -85,B 0,C 180,E1 -9794.889,E2 -9794.889} C_VEL
LIN {X 0,Y 427.234,Z 347.919,A -85,B 0,C 180,E1 -9795.813,E2 -9795.813} C_VEL
LIN {X 0,Y 426.55,Z 358.881,A -85,B 0,C 180,E1 -9796.906,E2 -9796.906} C_VEL
LIN {X 0,Y 425.947,Z 368.542,A -85,B 0,C 180,E1 -9798.098,E2 -9798.098} C_VEL
LIN {X 0,Y 425.39,Z 376.465,A -85,B 0,C 180,E1 -9799.289,E2 -9799.289} C_VEL
LIN {X 0,Y 424.902,Z 384.21,A -85,B 0,C 180,E1 -9800.72,E2 -9800.72} C_VEL
LIN {X 0,Y 424.465,Z 391.354,A -85,B 0,C 180,E1 -9802.388,E2 -9802.388} C_VEL
LIN {X 0,Y 424.277,Z 396.495,A -85,B 0,C 180,E1 -9803.945,E2 -9803.945} C_VEL
LIN {X 0,Y 424.226,Z 399.759,A -85,B 0,C 180,E1 -9805.249,E2 -9805.249} C_VEL
LIN {X 0,Y 424.12,Z 401.633,A -85,B 0,C 180,E1 -9806.2,E2 -9806.2} C_VEL
LIN {X 0,Y 424.192,Z 403.049,A -85,B 0,C 180,E1 -9807.151,E2 -9807.151} C_VEL
LIN {X 0,Y 424.115,Z 404.665,A -85,B 0,C 180,E1 -9809.051,E2 -9809.051} C_VEL
LIN {X 0,Y 424.13,Z 404.885,A -85,B 0,C 180,E1 -9810,E2 -9810} C_VEL
LIN {X 0,Y 424.115,Z 404.666,A -85,B 0,C 180,E1 -9810.95,E2 -9810.95} C_VEL
LIN {X 0,Y 424.192,Z 403.052,A -85,B 0,C 180,E1 -9812.849,E2 -9812.849} C_VEL
LIN {X 0,Y 424.12,Z 401.637,A -85,B 0,C 180,E1 -9813.801,E2 -9813.801} C_VEL
LIN {X 0,Y 424.28,Z 398.68,A -85,B 0,C 180,E1 -9815.227,E2 -9815.227} C_VEL
LIN {X 0,Y 424.36,Z 394.67,A -85,B 0,C 180,E1 -9816.657,E2 -9816.657} C_VEL
LIN {X 0,Y 424.651,Z 388.515,A -85,B 0,C 180,E1 -9818.327,E2 -9818.327} C_VEL
LIN {X 0,Y 425.047,Z 381.796,A -85,B 0,C 180,E1 -9819.758,E2 -9819.758} C_VEL
LIN {X 0,Y 425.582,Z 373.465,A -85,B 0,C 180,E1 -9821.189,E2 -9821.189} C_VEL
LIN {X 0,Y 426.214,Z 364.938,A -85,B 0,C 180,E1 -9822.378,E2 -9822.378} C_VEL
LIN {X 0,Y 426.831,Z 355.475,A -85,B 0,C 180,E1 -9823.46,E2 -9823.46} C_VEL
LIN {X 0,Y 427.471,Z 343.987,A -85,B 0,C 180,E1 -9824.521,E2 -9824.521} C_VEL
LIN {X 0,Y 428.238,Z 332.587,A -85,B 0,C 180,E1 -9825.345,E2 -9825.345} C_VEL
LIN {X 0,Y 428.641,Z 322.101,A -85,B 0,C 180,E1 -9825.94,E2 -9825.94} C_VEL
LIN {X 0,Y 426.777,Z 309.24,A -85,B 0,C 180,E1 -9826.56,E2 -9826.56} C_VEL
LIN {X 0,Y 424.788,Z 296.707,A -85,B 0,C 180,E1 -9827.008,E2 -9827.008} C_VEL
LIN {X 0,Y 425.108,Z 290.118,A -85,B 0,C 180,E1 -9829.551,E2 -9829.551} C_VEL
LIN {X 0,Y 425.47,Z 281.562,A -85,B 0,C 180,E1 -9832.841,E2 -9832.841} C_VEL
LIN {X 0,Y 425.903,Z 273.56,A -85,B 0,C 180,E1 -9835.931,E2 -9835.931} C_VEL
LIN {X 0,Y 426.348,Z 265.454,A -85,B 0,C 180,E1 -9839.113,E2 -9839.113} C_VEL
LIN {X 0,Y 426.882,Z 257.493,A -85,B 0,C 180,E1 -9842.349,E2 -9842.349} C_VEL
LIN {X 0,Y 427.375,Z 250.907,A -85,B 0,C 180,E1 -9845.139,E2 -9845.139} C_VEL
LIN {X 0,Y 427.302,Z 246.962,A -85,B 0,C 180,E1 -9846.893,E2 -9846.893} C_VEL
LIN {X 0,Y 426.226,Z 240.439,A -85,B 0,C 180,E1 -9850.021,E2 -9850.021} C_VEL
LIN {X 0,Y 425.331,Z 235.51,A -85,B 0,C 180,E1 -9852.553,E2 -9852.553} C_VEL
LIN {X 0,Y 425.261,Z 235.513,A -85,B 0,C 180,E1 -9856.044,E2 -9856.044} C_VEL
LIN {X 0,Y 425.254,Z 235.515,A -85,B 0,C 180,E1 -9858.619,E2 -9858.619} C_VEL
LIN {X 0,Y 425.283,Z 235.509,A -85,B 0,C 180,E1 -9861.1,E2 -9861.1} C_VEL
LIN {X 0,Y 425.302,Z 235.509,A -85,B 0,C 180,E1 -9864.664,E2 -9864.664} C_VEL
LIN {X 0,Y 425.269,Z 235.513,A -85,B 0,C 180,E1 -9868.073,E2 -9868.073} C_VEL
LIN {X 0,Y 425.308,Z 235.505,A -85,B 0,C 180,E1 -9871.366,E2 -9871.366} C_VEL
LIN {X 0,Y 425.263,Z 235.513,A -85,B 0,C 180,E1 -9874.553,E2 -9874.553} C_VEL
LIN {X 0,Y 425.296,Z 235.509,A -85,B 0,C 180,E1 -9877.73,E2 -9877.73} C_VEL
LIN {X 0,Y 425.366,Z 235.499,A -85,B 0,C 180,E1 -9880.704,E2 -9880.704} C_VEL
LIN {X 0,Y 425.392,Z 235.497,A -85,B 0,C 180,E1 -9883.688,E2 -9883.688} C_VEL
LIN {X 0,Y 425.413,Z 235.494,A -85,B 0,C 180,E1 -9887.598,E2 -9887.598} C_VEL
LIN {X 0,Y 425.409,Z 235.496,A -85,B 0,C 180,E1 -9891.449,E2 -9891.449} C_VEL
LIN {X 0,Y 425.553,Z 235.476,A -85,B 0,C 180,E1 -9894.313,E2 -9894.313} C_VEL
LIN {X 0,Y 425.577,Z 235.473,A -85,B 0,C 180,E1 -9898.107,E2 -9898.107} C_VEL
LIN {X 0,Y 425.577,Z 235.473,A -85,B 0,C 180,E1 -9900,E2 -9900} C_VEL
LIN {X 0,Y 425.528,Z 235.478,A -85,B 0,C 180,E1 -9902.84,E2 -9902.84} C_VEL
LIN {X 0,Y 425.549,Z 235.477,A -85,B 0,C 180,E1 -9905.687,E2 -9905.687} C_VEL
LIN {X 0,Y 425.413,Z 235.493,A -85,B 0,C 180,E1 -9908.551,E2 -9908.551} C_VEL
LIN {X 0,Y 425.417,Z 235.492,A -85,B 0,C 180,E1 -9912.402,E2 -9912.402} C_VEL
LIN {X 0,Y 425.388,Z 235.495,A -85,B 0,C 180,E1 -9916.312,E2 -9916.312} C_VEL
LIN {X 0,Y 425.333,Z 235.502,A -85,B 0,C 180,E1 -9919.635,E2 -9919.635} C_VEL
LIN {X 0,Y 425.292,Z 235.509,A -85,B 0,C 180,E1 -9922.339,E2 -9922.339} C_VEL
LIN {X 0,Y 425.325,Z 235.506,A -85,B 0,C 180,E1 -9924.657,E2 -9924.657} C_VEL
LIN {X 0,Y 425.27,Z 235.51,A -85,B 0,C 180,E1 -9927.563,E2 -9927.563} C_VEL
LIN {X 0,Y 425.29,Z 235.509,A -85,B 0,C 180,E1 -9930.816,E2 -9930.816} C_VEL
LIN {X 0,Y 425.314,Z 235.509,A -85,B 0,C 180,E1 -9934.287,E2 -9934.287} C_VEL
LIN {X 0,Y 425.281,Z 235.51,A -85,B 0,C 180,E1 -9937.694,E2 -9937.694} C_VEL
LIN {X 0,Y 425.28,Z 235.512,A -85,B 0,C 180,E1 -9940.52,E2 -9940.52} C_VEL
LIN {X 0,Y 425.264,Z 235.514,A -85,B 0,C 180,E1 -9943.956,E2 -9943.956} C_VEL
LIN {X 0,Y 425.273,Z 235.509,A -85,B 0,C 180,E1 -9947.346,E2 -9947.346} C_VEL
LIN {X 0,Y 425.287,Z 235.512,A -85,B 0,C 180,E1 -9949.872,E2 -9949.872} C_VEL
LIN {X 0,Y 425.275,Z 235.51,A -85,B 0,C 180,E1 -9952.489,E2 -9952.489} C_VEL
LIN {X 0,Y 425.122,Z 235.533,A -85,B 0,C 180,E1 -9955.75,E2 -9955.75} C_VEL
LIN {X 0,Y 424.801,Z 235.573,A -85,B 0,C 180,E1 -9958.034,E2 -9958.034} C_VEL
LIN {X 0,Y 424.714,Z 238.536,A -85,B 0,C 180,E1 -9961.322,E2 -9961.322} C_VEL
LIN {X 0,Y 424.61,Z 241.622,A -85,B 0,C 180,E1 -9964.51,E2 -9964.51} C_VEL
LIN {X 0,Y 424.523,Z 244.74,A -85,B 0,C 180,E1 -9967.619,E2 -9967.619} C_VEL
LIN {X 0,Y 424.543,Z 247.963,A -85,B 0,C 180,E1 -9970.665,E2 -9970.665} C_VEL
LIN {X 0,Y 424.534,Z 250.749,A -85,B 0,C 180,E1 -9973.11,E2 -9973.11} C_VEL
LIN {X 0,Y 428.007,Z 264.496,A -85,B 0,C 180,E1 -9973.714,E2 -9973.714} C_VEL
LIN {X 0,Y 429.385,Z 271.487,A -85,B 0,C 180,E1 -9974.088,E2 -9974.088} C_VEL
LIN {X 0,Y 428.768,Z 283.878,A -85,B 0,C 180,E1 -9974.796,E2 -9974.796} C_VEL
LIN {X 0,Y 428.237,Z 294.72,A -85,B 0,C 180,E1 -9975.607,E2 -9975.607} C_VEL
LIN {X 0,Y 427.605,Z 305.078,A -85,B 0,C 180,E1 -9976.576,E2 -9976.576} C_VEL
LIN {X 0,Y 426.941,Z 314.374,A -85,B 0,C 180,E1 -9977.643,E2 -9977.643} C_VEL
LIN {X 0,Y 426.376,Z 322.837,A -85,B 0,C 180,E1 -9978.832,E2 -9978.832} C_VEL
LIN {X 0,Y 425.77,Z 331.053,A -85,B 0,C 180,E1 -9980.259,E2 -9980.259} C_VEL
LIN {X 0,Y 425.318,Z 336.675,A -85,B 0,C 180,E1 -9981.447,E2 -9981.447} C_VEL
LIN {X 0,Y 424.981,Z 342.083,A -85,B 0,C 180,E1 -9982.856,E2 -9982.856} C_VEL
LIN {X 0,Y 424.594,Z 346.447,A -85,B 0,C 180,E1 -9984.3,E2 -9984.3} C_VEL
LIN {X 0,Y 424.569,Z 348.711,A -85,B 0,C 180,E1 -9985.252,E2 -9985.252} C_VEL
LIN {X 0,Y 424.523,Z 350.556,A -85,B 0,C 180,E1 -9986.203,E2 -9986.203} C_VEL
LIN {X 0,Y 424.408,Z 351.951,A -85,B 0,C 180,E1 -9987.152,E2 -9987.152} C_VEL
LIN {X 0,Y 424.246,Z 353.555,A -85,B 0,C 180,E1 -9989.051,E2 -9989.051} C_VEL
LIN {X 0,Y 424.234,Z 353.788,A -85,B 0,C 180,E1 -9990,E2 -9990} C_VEL
LIN {X 0,Y 424.246,Z 353.464,A -85,B 0,C 180,E1 -9991.173,E2 -9991.173} C_VEL
LIN {X 0,Y 423.606,Z 353.025,A -85,B 0,C 180,E1 -9991.966,E2 -9991.966} C_VEL
LIN {X 0,Y 420.82,Z 351.813,A -85,B 0,C 180,E1 -9993.253,E2 -9993.253} C_VEL
LIN {X 0,Y 418.493,Z 350.404,A -85,B 0,C 180,E1 -9994.278,E2 -9994.278} C_VEL
LIN {X 0,Y 417.536,Z 348.901,A -85,B 0,C 180,E1 -9995.055,E2 -9995.055} C_VEL
LIN {X 0,Y 417.481,Z 348.297,A -85,B 0,C 180,E1 -9995.314,E2 -9995.314} C_VEL
LIN {X 0,Y 417.817,Z 344.435,A -85,B 0,C 180,E1 -9996.762,E2 -9996.762} C_VEL
LIN {X 0,Y 418.126,Z 339.456,A -85,B 0,C 180,E1 -9998.214,E2 -9998.214} C_VEL
LIN {X 0,Y 418.63,Z 333.178,A -85,B 0,C 180,E1 -9999.665,E2 -9999.665} C_VEL
LIN {X 0,Y 419.266,Z 325.315,A -85,B 0,C 180,E1 -10001.114,E2 -10001.114} C_VEL
LIN {X 0,Y 419.876,Z 317.296,A -85,B 0,C 180,E1 -10002.322,E2 -10002.322} C_VEL
LIN {X 0,Y 420.642,Z 307.5,A -85,B 0,C 180,E1 -10003.527,E2 -10003.527} C_VEL
LIN {X 0,Y 421.224,Z 297.863,A -85,B 0,C 180,E1 -10004.493,E2 -10004.493} C_VEL
LIN {X 0,Y 421.853,Z 287.426,A -85,B 0,C 180,E1 -10005.336,E2 -10005.336} C_VEL
LIN {X 0,Y 422.425,Z 274.846,A -85,B 0,C 180,E1 -10006.119,E2 -10006.119} C_VEL
LIN {X 0,Y 422.434,Z 271.363,A -85,B 0,C 180,E1 -10006.305,E2 -10006.305} C_VEL
LIN {X 0,Y 419.58,Z 259.037,A -85,B 0,C 180,E1 -10006.949,E2 -10006.949} C_VEL
LIN {X 0,Y 417.46,Z 251.112,A -85,B 0,C 180,E1 -10007.286,E2 -10007.286} C_VEL
LIN {X 0,Y 417.46,Z 248.463,A -85,B 0,C 180,E1 -10009.676,E2 -10009.676} C_VEL
LIN {X 0,Y 417.467,Z 245.216,A -85,B 0,C 180,E1 -10012.78,E2 -10012.78} C_VEL
LIN {X 0,Y 417.567,Z 243.092,A -85,B 0,C 180,E1 -10014.883,E2 -10014.883} C_VEL
LIN {X 0,Y 417.644,Z 239.994,A -85,B 0,C 180,E1 -10018.111,E2 -10018.111} C_VEL
LIN {X 0,Y 417.726,Z 236.862,A -85,B 0,C 180,E1 -10021.437,E2 -10021.437} C_VEL
LIN {X 0,Y 417.851,Z 236.44,A -85,B 0,C 180,E1 -10022.757,E2 -10022.757} C_VEL
LIN {X 0,Y 418.114,Z 236.402,A -85,B 0,C 180,E1 -10024.855,E2 -10024.855} C_VEL
LIN {X 0,Y 418.224,Z 236.39,A -85,B 0,C 180,E1 -10027.832,E2 -10027.832} C_VEL
LIN {X 0,Y 418.221,Z 236.387,A -85,B 0,C 180,E1 -10030.948,E2 -10030.948} C_VEL
LIN {X 0,Y 418.21,Z 236.391,A -85,B 0,C 180,E1 -10033.729,E2 -10033.729} C_VEL
LIN {X 0,Y 418.209,Z 236.391,A -85,B 0,C 180,E1 -10036.448,E2 -10036.448} C_VEL
LIN {X 0,Y 418.223,Z 236.388,A -85,B 0,C 180,E1 -10039.131,E2 -10039.131} C_VEL
LIN {X 0,Y 418.227,Z 236.39,A -85,B 0,C 180,E1 -10042.167,E2 -10042.167} C_VEL
LIN {X 0,Y 418.266,Z 236.385,A -85,B 0,C 180,E1 -10045.42,E2 -10045.42} C_VEL
LIN {X 0,Y 418.213,Z 236.387,A -85,B 0,C 180,E1 -10048.604,E2 -10048.604} C_VEL
LIN {X 0,Y 418.223,Z 236.389,A -85,B 0,C 180,E1 -10051.931,E2 -10051.931} C_VEL
LIN {X 0,Y 418.274,Z 236.385,A -85,B 0,C 180,E1 -10055.162,E2 -10055.162} C_VEL
LIN {X 0,Y 418.237,Z 236.386,A -85,B 0,C 180,E1 -10058.304,E2 -10058.304} C_VEL
LIN {X 0,Y 418.276,Z 236.384,A -85,B 0,C 180,E1 -10061.383,E2 -10061.383} C_VEL
LIN {X 0,Y 418.294,Z 236.378,A -85,B 0,C 180,E1 -10064.406,E2 -10064.406} C_VEL
LIN {X 0,Y 418.359,Z 236.373,A -85,B 0,C 180,E1 -10067.386,E2 -10067.386} C_VEL
LIN {X 0,Y 418.344,Z 236.374,A -85,B 0,C 180,E1 -10070.329,E2 -10070.329} C_VEL
LIN {X 0,Y 418.516,Z 236.353,A -85,B 0,C 180,E1 -10072.279,E2 -10072.279} C_VEL
LIN {X 0,Y 418.51,Z 236.353,A -85,B 0,C 180,E1 -10074.217,E2 -10074.217} C_VEL
LIN {X 0,Y 418.539,Z 236.348,A -85,B 0,C 180,E1 -10078.075,E2 -10078.075} C_VEL
LIN {X 0,Y 418.484,Z 236.357,A -85,B 0,C 180,E1 -10080.962,E2 -10080.962} C_VEL
LIN {X 0,Y 418.503,Z 236.355,A -85,B 0,C 180,E1 -10082.888,E2 -10082.888} C_VEL
LIN {X 0,Y 418.509,Z 236.353,A -85,B 0,C 180,E1 -10085.783,E2 -10085.783} C_VEL
LIN {X 0,Y 418.378,Z 236.37,A -85,B 0,C 180,E1 -10088.696,E2 -10088.696} C_VEL
LIN {X 0,Y 418.306,Z 236.377,A -85,B 0,C 180,E1 -10091.631,E2 -10091.631} C_VEL
LIN {X 0,Y 418.302,Z 236.379,A -85,B 0,C 180,E1 -10094.597,E2 -10094.597} C_VEL
LIN {X 0,Y 418.291,Z 236.382,A -85,B 0,C 180,E1 -10097.604,E2 -10097.604} C_VEL
LIN {X 0,Y 418.253,Z 236.384,A -85,B 0,C 180,E1 -10100.663,E2 -10100.663} C_VEL
LIN {X 0,Y 418.261,Z 236.387,A -85,B 0,C 180,E1 -10103.783,E2 -10103.783} C_VEL
LIN {X 0,Y 418.21,Z 236.389,A -85,B 0,C 180,E1 -10107.043,E2 -10107.043} C_VEL
LIN {X 0,Y 418.243,Z 236.386,A -85,B 0,C 180,E1 -10110.272,E2 -10110.272} C_VEL
LIN {X 0,Y 418.25,Z 236.388,A -85,B 0,C 180,E1 -10113.677,E2 -10113.677} C_VEL
LIN {X 0,Y 418.239,Z 236.388,A -85,B 0,C 180,E1 -10117.224,E2 -10117.224} C_VEL
LIN {X 0,Y 418.209,Z 236.39,A -85,B 0,C 180,E1 -10120.867,E2 -10120.867} C_VEL
LIN {X 0,Y 418.206,Z 236.392,A -85,B 0,C 180,E1 -10123.729,E2 -10123.729} C_VEL
LIN {X 0,Y 418.286,Z 236.531,A -85,B 0,C 180,E1 -10127.174,E2 -10127.174} C_VEL
LIN {X 0,Y 419.431,Z 242.846,A -85,B 0,C 180,E1 -10130.452,E2 -10130.452} C_VEL
LIN {X 0,Y 420.391,Z 248.901,A -85,B 0,C 180,E1 -10133.365,E2 -10133.365} C_VEL
LIN {X 0,Y 420.303,Z 253.345,A -85,B 0,C 180,E1 -10135.353,E2 -10135.353} C_VEL
LIN {X 0,Y 419.711,Z 261.312,A -85,B 0,C 180,E1 -10138.729,E2 -10138.729} C_VEL
LIN {X 0,Y 419.203,Z 269.3,A -85,B 0,C 180,E1 -10142.003,E2 -10142.003} C_VEL
LIN {X 0,Y 418.674,Z 277.286,A -85,B 0,C 180,E1 -10145.187,E2 -10145.187} C_VEL
LIN {X 0,Y 418.286,Z 285.182,A -85,B 0,C 180,E1 -10148.306,E2 -10148.306} C_VEL
LIN {X 0,Y 417.926,Z 292.974,A -85,B 0,C 180,E1 -10151.367,E2 -10151.367} C_VEL
LIN {X 0,Y 417.735,Z 296.409,A -85,B 0,C 180,E1 -10152.713,E2 -10152.713} C_VEL
LIN {X 0,Y 419.987,Z 310.537,A -85,B 0,C 180,E1 -10153.226,E2 -10153.226} C_VEL
LIN {X 0,Y 421.753,Z 322.822,A -85,B 0,C 180,E1 -10153.855,E2 -10153.855} C_VEL
LIN {X 0,Y 421.1,Z 335.707,A -85,B 0,C 180,E1 -10154.636,E2 -10154.636} C_VEL
LIN {X 0,Y 420.386,Z 346.42,A -85,B 0,C 180,E1 -10155.477,E2 -10155.477} C_VEL
LIN {X 0,Y 419.655,Z 357.373,A -85,B 0,C 180,E1 -10156.564,E2 -10156.564} C_VEL
LIN {X 0,Y 419.115,Z 366.318,A -85,B 0,C 180,E1 -10157.655,E2 -10157.655} C_VEL
LIN {X 0,Y 418.382,Z 376.035,A -85,B 0,C 180,E1 -10159.107,E2 -10159.107} C_VEL
LIN {X 0,Y 417.86,Z 383.781,A -85,B 0,C 180,E1 -10160.562,E2 -10160.562} C_VEL
LIN {X 0,Y 417.539,Z 389.092,A -85,B 0,C 180,E1 -10161.774,E2 -10161.774} C_VEL
LIN {X 0,Y 417.278,Z 395.26,A -85,B 0,C 180,E1 -10163.57,E2 -10163.57} C_VEL
LIN {X 0,Y 417.162,Z 399.332,A -85,B 0,C 180,E1 -10165.168,E2 -10165.168} C_VEL
LIN {X 0,Y 417.035,Z 401.206,A -85,B 0,C 180,E1 -10166.135,E2 -10166.135} C_VEL
LIN {X 0,Y 417.106,Z 402.621,A -85,B 0,C 180,E1 -10167.103,E2 -10167.103} C_VEL
LIN {X 0,Y 417.035,Z 404.239,A -85,B 0,C 180,E1 -10169.035,E2 -10169.035} C_VEL
LIN {X 0,Y 417.047,Z 404.458,A -85,B 0,C 180,E1 -10170,E2 -10170} C_VEL
LIN {X 0,Y 417.035,Z 404.239,A -85,B 0,C 180,E1 -10170.966,E2 -10170.966} C_VEL
LIN {X 0,Y 417.107,Z 402.624,A -85,B 0,C 180,E1 -10172.898,E2 -10172.898} C_VEL
LIN {X 0,Y 417.035,Z 401.209,A -85,B 0,C 180,E1 -10173.865,E2 -10173.865} C_VEL
LIN {X 0,Y 417.193,Z 398.252,A -85,B 0,C 180,E1 -10175.316,E2 -10175.316} C_VEL
LIN {X 0,Y 417.276,Z 394.241,A -85,B 0,C 180,E1 -10176.771,E2 -10176.771} C_VEL
LIN {X 0,Y 417.589,Z 388.085,A -85,B 0,C 180,E1 -10178.468,E2 -10178.468} C_VEL
LIN {X 0,Y 418.015,Z 381.366,A -85,B 0,C 180,E1 -10179.924,E2 -10179.924} C_VEL
LIN {X 0,Y 418.595,Z 373.036,A -85,B 0,C 180,E1 -10181.378,E2 -10181.378} C_VEL
LIN {X 0,Y 419.214,Z 364.506,A -85,B 0,C 180,E1 -10182.588,E2 -10182.588} C_VEL
LIN {X 0,Y 419.956,Z 353.581,A -85,B 0,C 180,E1 -10183.838,E2 -10183.838} C_VEL
LIN {X 0,Y 420.67,Z 342.124,A -85,B 0,C 180,E1 -10184.884,E2 -10184.884} C_VEL
LIN {X 0,Y 421.486,Z 330.229,A -85,B 0,C 180,E1 -10185.722,E2 -10185.722} C_VEL
LIN {X 0,Y 421.726,Z 322.804,A -85,B 0,C 180,E1 -10186.147,E2 -10186.147} C_VEL
LIN {X 0,Y 419.894,Z 309.759,A -85,B 0,C 180,E1 -10186.807,E2 -10186.807} C_VEL
LIN {X 0,Y 417.735,Z 296.357,A -85,B 0,C 180,E1 -10187.287,E2 -10187.287} C_VEL
LIN {X 0,Y 418.062,Z 289.095,A -85,B 0,C 180,E1 -10190.159,E2 -10190.159} C_VEL
LIN {X 0,Y 418.483,Z 281.238,A -85,B 0,C 180,E1 -10193.245,E2 -10193.245} C_VEL
LIN {X 0,Y 418.931,Z 273.257,A -85,B 0,C 180,E1 -10196.396,E2 -10196.396} C_VEL
LIN {X 0,Y 419.358,Z 265.838,A -85,B 0,C 180,E1 -10199.37,E2 -10199.37} C_VEL
LIN {X 0,Y 419.889,Z 258.599,A -85,B 0,C 180,E1 -10202.386,E2 -10202.386} C_VEL
LIN {X 0,Y 420.378,Z 252.523,A -85,B 0,C 180,E1 -10204.995,E2 -10204.995} C_VEL
LIN {X 0,Y 420.305,Z 248.057,A -85,B 0,C 180,E1 -10207.011,E2 -10207.011} C_VEL
LIN {X 0,Y 419.234,Z 241.541,A -85,B 0,C 180,E1 -10210.196,E2 -10210.196} C_VEL
LIN {X 0,Y 418.262,Z 236.391,A -85,B 0,C 180,E1 -10212.906,E2 -10212.906} C_VEL
LIN {X 0,Y 418.207,Z 236.391,A -85,B 0,C 180,E1 -10216.272,E2 -10216.272} C_VEL
LIN {X 0,Y 418.211,Z 236.39,A -85,B 0,C 180,E1 -10219.133,E2 -10219.133} C_VEL
LIN {X 0,Y 418.241,Z 236.388,A -85,B 0,C 180,E1 -10222.776,E2 -10222.776} C_VEL
LIN {X 0,Y 418.252,Z 236.388,A -85,B 0,C 180,E1 -10226.323,E2 -10226.323} C_VEL
LIN {X 0,Y 418.245,Z 236.385,A -85,B 0,C 180,E1 -10229.728,E2 -10229.728} C_VEL
LIN {X 0,Y 418.214,Z 236.388,A -85,B 0,C 180,E1 -10233.017,E2 -10233.017} C_VEL
LIN {X 0,Y 418.263,Z 236.387,A -85,B 0,C 180,E1 -10236.217,E2 -10236.217} C_VEL
LIN {X 0,Y 418.254,Z 236.384,A -85,B 0,C 180,E1 -10239.337,E2 -10239.337} C_VEL
LIN {X 0,Y 418.29,Z 236.382,A -85,B 0,C 180,E1 -10242.396,E2 -10242.396} C_VEL
LIN {X 0,Y 418.304,Z 236.379,A -85,B 0,C 180,E1 -10245.403,E2 -10245.403} C_VEL
LIN {X 0,Y 418.306,Z 236.377,A -85,B 0,C 180,E1 -10248.369,E2 -10248.369} C_VEL
LIN {X 0,Y 418.47,Z 236.358,A -85,B 0,C 180,E1 -10252.279,E2 -10252.279} C_VEL
LIN {X 0,Y 418.511,Z 236.353,A -85,B 0,C 180,E1 -10254.217,E2 -10254.217} C_VEL
LIN {X 0,Y 418.546,Z 236.349,A -85,B 0,C 180,E1 -10258.076,E2 -10258.076} C_VEL
LIN {X 0,Y 418.411,Z 236.365,A -85,B 0,C 180,E1 -10260.962,E2 -10260.962} C_VEL
LIN {X 0,Y 418.485,Z 236.355,A -85,B 0,C 180,E1 -10262.888,E2 -10262.888} C_VEL
LIN {X 0,Y 418.474,Z 236.357,A -85,B 0,C 180,E1 -10266.647,E2 -10266.647} C_VEL
LIN {X 0,Y 418.344,Z 236.374,A -85,B 0,C 180,E1 -10269.671,E2 -10269.671} C_VEL
LIN {X 0,Y 418.351,Z 236.375,A -85,B 0,C 180,E1 -10273.001,E2 -10273.001} C_VEL
LIN {X 0,Y 418.316,Z 236.379,A -85,B 0,C 180,E1 -10276.734,E2 -10276.734} C_VEL
LIN {X 0,Y 418.275,Z 236.381,A -85,B 0,C 180,E1 -10279.79,E2 -10279.79} C_VEL
LIN {X 0,Y 418.236,Z 236.39,A -85,B 0,C 180,E1 -10282.736,E2 -10282.736} C_VEL
LIN {X 0,Y 418.24,Z 236.386,A -85,B 0,C 180,E1 -10285.906,E2 -10285.906} C_VEL
LIN {X 0,Y 418.262,Z 236.383,A -85,B 0,C 180,E1 -10289.162,E2 -10289.162} C_VEL
LIN {X 0,Y 418.261,Z 236.384,A -85,B 0,C 180,E1 -10292.844,E2 -10292.844} C_VEL
LIN {X 0,Y 418.248,Z 236.389,A -85,B 0,C 180,E1 -10296.238,E2 -10296.238} C_VEL
LIN {X 0,Y 418.246,Z 236.386,A -85,B 0,C 180,E1 -10299.683,E2 -10299.683} C_VEL
LIN {X 0,Y 418.227,Z 236.392,A -85,B 0,C 180,E1 -10302.32,E2 -10302.32} C_VEL
LIN {X 0,Y 418.239,Z 236.384,A -85,B 0,C 180,E1 -10305.109,E2 -10305.109} C_VEL
LIN {X 0,Y 418.237,Z 236.389,A -85,B 0,C 180,E1 -10307.766,E2 -10307.766} C_VEL
LIN {X 0,Y 418.245,Z 236.385,A -85,B 0,C 180,E1 -10310.621,E2 -10310.621} C_VEL
LIN {X 0,Y 418.183,Z 236.396,A -85,B 0,C 180,E1 -10313.969,E2 -10313.969} C_VEL
LIN {X 0,Y 417.959,Z 236.423,A -85,B 0,C 180,E1 -10316.296,E2 -10316.296} C_VEL
LIN {X 0,Y 417.714,Z 236.781,A -85,B 0,C 180,E1 -10318.562,E2 -10318.562} C_VEL
LIN {X 0,Y 417.646,Z 239.886,A -85,B 0,C 180,E1 -10321.889,E2 -10321.889} C_VEL
LIN {X 0,Y 417.572,Z 243.219,A -85,B 0,C 180,E1 -10325.348,E2 -10325.348} C_VEL
LIN {X 0,Y 417.481,Z 246.182,A -85,B 0,C 180,E1 -10328.262,E2 -10328.262} C_VEL
LIN {X 0,Y 417.454,Z 249.513,A -85,B 0,C 180,E1 -10331.345,E2 -10331.345} C_VEL
LIN {X 0,Y 417.465,Z 251.15,A -85,B 0,C 180,E1 -10332.802,E2 -10332.802} C_VEL
LIN {X 0,Y 421.219,Z 265.69,A -85,B 0,C 180,E1 -10333.475,E2 -10333.475} C_VEL
LIN {X 0,Y 422.54,Z 272.644,A -85,B 0,C 180,E1 -10333.86,E2 -10333.86} C_VEL
LIN {X 0,Y 421.958,Z 284.31,A -85,B 0,C 180,E1 -10334.544,E2 -10334.544} C_VEL
LIN {X 0,Y 421.286,Z 296.801,A -85,B 0,C 180,E1 -10335.508,E2 -10335.508} C_VEL
LIN {X 0,Y 420.656,Z 306.664,A -85,B 0,C 180,E1 -10336.473,E2 -10336.473} C_VEL
LIN {X 0,Y 419.907,Z 316.608,A -85,B 0,C 180,E1 -10337.678,E2 -10337.678} C_VEL
LIN {X 0,Y 419.327,Z 324.738,A -85,B 0,C 180,E1 -10338.887,E2 -10338.887} C_VEL
LIN {X 0,Y 418.671,Z 332.702,A -85,B 0,C 180,E1 -10340.336,E2 -10340.336} C_VEL
LIN {X 0,Y 418.184,Z 339.09,A -85,B 0,C 180,E1 -10341.787,E2 -10341.787} C_VEL
LIN {X 0,Y 417.882,Z 344.151,A -85,B 0,C 180,E1 -10343.239,E2 -10343.239} C_VEL
LIN {X 0,Y 417.507,Z 348.089,A -85,B 0,C 180,E1 -10344.688,E2 -10344.688} C_VEL
LIN {X 0,Y 417.467,Z 350.983,A -85,B 0,C 180,E1 -10346.139,E2 -10346.139} C_VEL
LIN {X 0,Y 417.341,Z 352.378,A -85,B 0,C 180,E1 -10347.104,E2 -10347.104} C_VEL
LIN {X 0,Y 417.161,Z 353.982,A -85,B 0,C 180,E1 -10349.035,E2 -10349.035} C_VEL
LIN {X 0,Y 417.16,Z 354.214,A -85,B 0,C 180,E1 -10350,E2 -10350} C_VEL
LIN {X 0,Y 417.214,Z 353.447,A -85,B 0,C 180,E1 -10351.931,E2 -10351.931} C_VEL
LIN {X 0,Y 417.464,Z 351.135,A -85,B 0,C 180,E1 -10353.861,E2 -10353.861} C_VEL
LIN {X 0,Y 417.481,Z 348.297,A -85,B 0,C 180,E1 -10355.314,E2 -10355.314} C_VEL
LIN {X 0,Y 416.919,Z 346.463,A -85,B 0,C 180,E1 -10356.08,E2 -10356.08} C_VEL
LIN {X 0,Y 414.307,Z 343.077,A -85,B 0,C 180,E1 -10357.319,E2 -10357.319} C_VEL
LIN {X 0,Y 411.805,Z 339.12,A -85,B 0,C 180,E1 -10358.533,E2 -10358.533} C_VEL
LIN {X 0,Y 411.417,Z 336.229,A -85,B 0,C 180,E1 -10359.249,E2 -10359.249} C_VEL
LIN {X 0,Y 412.048,Z 328.547,A -85,B 0,C 180,E1 -10360.814,E2 -10360.814} C_VEL
LIN {X 0,Y 412.878,Z 319.48,A -85,B 0,C 180,E1 -10362.285,E2 -10362.285} C_VEL
LIN {X 0,Y 413.58,Z 310.046,A -85,B 0,C 180,E1 -10363.512,E2 -10363.512} C_VEL
LIN {X 0,Y 414.275,Z 300.08,A -85,B 0,C 180,E1 -10364.566,E2 -10364.566} C_VEL
LIN {X 0,Y 414.941,Z 289.456,A -85,B 0,C 180,E1 -10365.471,E2 -10365.471} C_VEL
LIN {X 0,Y 415.524,Z 278.984,A -85,B 0,C 180,E1 -10366.177,E2 -10366.177} C_VEL
LIN {X 0,Y 415.645,Z 272.745,A -85,B 0,C 180,E1 -10366.53,E2 -10366.53} C_VEL
LIN {X 0,Y 412.843,Z 260.653,A -85,B 0,C 180,E1 -10367.192,E2 -10367.192} C_VEL
LIN {X 0,Y 410.418,Z 251.517,A -85,B 0,C 180,E1 -10367.601,E2 -10367.601} C_VEL
LIN {X 0,Y 410.416,Z 247.768,A -85,B 0,C 180,E1 -10371.076,E2 -10371.076} C_VEL
LIN {X 0,Y 410.53,Z 243.912,A -85,B 0,C 180,E1 -10374.861,E2 -10374.861} C_VEL
LIN {X 0,Y 410.603,Z 240.31,A -85,B 0,C 180,E1 -10378.637,E2 -10378.637} C_VEL
LIN {X 0,Y 410.686,Z 237.946,A -85,B 0,C 180,E1 -10381.169,E2 -10381.169} C_VEL
LIN {X 0,Y 410.72,Z 237.327,A -85,B 0,C 180,E1 -10382.036,E2 -10382.036} C_VEL
LIN {X 0,Y 411.076,Z 237.279,A -85,B 0,C 180,E1 -10384.851,E2 -10384.851} C_VEL
LIN {X 0,Y 411.199,Z 237.266,A -85,B 0,C 180,E1 -10388.167,E2 -10388.167} C_VEL
LIN {X 0,Y 411.162,Z 237.267,A -85,B 0,C 180,E1 -10391.228,E2 -10391.228} C_VEL
LIN {X 0,Y 411.177,Z 237.266,A -85,B 0,C 180,E1 -10394.49,E2 -10394.49} C_VEL
LIN {X 0,Y 411.175,Z 237.268,A -85,B 0,C 180,E1 -10398.194,E2 -10398.194} C_VEL
LIN {X 0,Y 411.21,Z 237.261,A -85,B 0,C 180,E1 -10400.775,E2 -10400.775} C_VEL
LIN {X 0,Y 411.199,Z 237.262,A -85,B 0,C 180,E1 -10404.471,E2 -10404.471} C_VEL
LIN {X 0,Y 411.209,Z 237.261,A -85,B 0,C 180,E1 -10406.873,E2 -10406.873} C_VEL
LIN {X 0,Y 411.213,Z 237.26,A -85,B 0,C 180,E1 -10410.65,E2 -10410.65} C_VEL
LIN {X 0,Y 411.189,Z 237.267,A -85,B 0,C 180,E1 -10413.616,E2 -10413.616} C_VEL
LIN {X 0,Y 411.198,Z 237.265,A -85,B 0,C 180,E1 -10416.852,E2 -10416.852} C_VEL
LIN {X 0,Y 411.217,Z 237.26,A -85,B 0,C 180,E1 -10420.051,E2 -10420.051} C_VEL
LIN {X 0,Y 411.265,Z 237.259,A -85,B 0,C 180,E1 -10423.131,E2 -10423.131} C_VEL
LIN {X 0,Y 411.308,Z 237.253,A -85,B 0,C 180,E1 -10426.896,E2 -10426.896} C_VEL
LIN {X 0,Y 411.296,Z 237.251,A -85,B 0,C 180,E1 -10430.161,E2 -10430.161} C_VEL
LIN {X 0,Y 411.485,Z 237.227,A -85,B 0,C 180,E1 -10432.147,E2 -10432.147} C_VEL
LIN {X 0,Y 411.473,Z 237.229,A -85,B 0,C 180,E1 -10434.118,E2 -10434.118} C_VEL
LIN {X 0,Y 411.508,Z 237.224,A -85,B 0,C 180,E1 -10438.042,E2 -10438.042} C_VEL
LIN {X 0,Y 411.448,Z 237.233,A -85,B 0,C 180,E1 -10440.979,E2 -10440.979} C_VEL
LIN {X 0,Y 411.46,Z 237.232,A -85,B 0,C 180,E1 -10442.937,E2 -10442.937} C_VEL
LIN {X 0,Y 411.47,Z 237.23,A -85,B 0,C 180,E1 -10445.882,E2 -10445.882} C_VEL
LIN {X 0,Y 411.318,Z 237.248,A -85,B 0,C 180,E1 -10448.846,E2 -10448.846} C_VEL
LIN {X 0,Y 411.277,Z 237.254,A -85,B 0,C 180,E1 -10451.833,E2 -10451.833} C_VEL
LIN {X 0,Y 411.26,Z 237.255,A -85,B 0,C 180,E1 -10454.853,E2 -10454.853} C_VEL
LIN {X 0,Y 411.255,Z 237.259,A -85,B 0,C 180,E1 -10457.915,E2 -10457.915} C_VEL
LIN {X 0,Y 411.199,Z 237.262,A -85,B 0,C 180,E1 -10461.034,E2 -10461.034} C_VEL
LIN {X 0,Y 411.194,Z 237.265,A -85,B 0,C 180,E1 -10464.217,E2 -10464.217} C_VEL
LIN {X 0,Y 411.173,Z 237.269,A -85,B 0,C 180,E1 -10467.484,E2 -10467.484} C_VEL
LIN {X 0,Y 411.198,Z 237.266,A -85,B 0,C 180,E1 -10469.713,E2 -10469.713} C_VEL
